Universal Robots URScript: samho_main_Fillet_2024_03_05.script

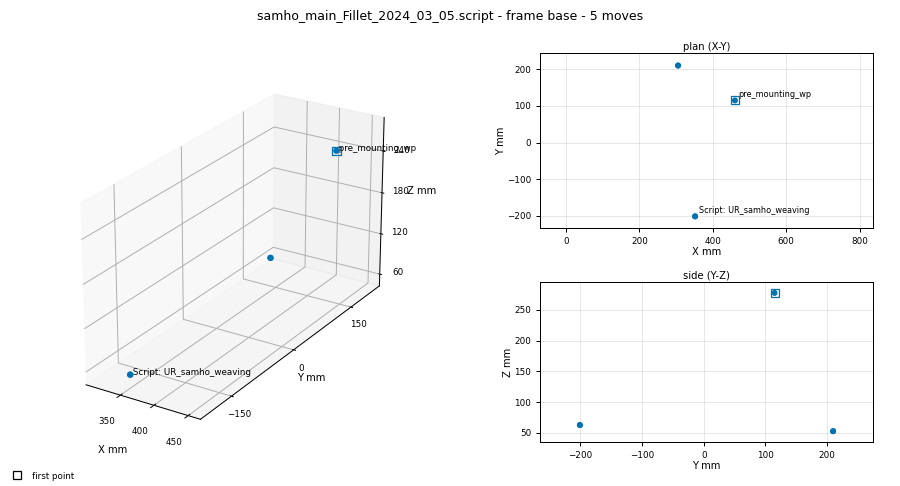
[picture p0: tool path of samho_main_Fillet_2024_03_05.script in frame base, 5 of 126 moves have a stored position in this frame; points joined in program order, loops and branches not executed]
def samho_main_Fillet_2024_03_05():
  modbus_add_signal("127.0.0.1", 255, 239, 2, "MODBUS_1", False)
  modbus_set_signal_update_frequency("MODBUS_1", 1)
  modbus_add_signal("127.0.0.1", 255, 153, 2, "MODBUS_2", False)
  modbus_set_signal_update_frequency("MODBUS_2", 10)
  modbus_add_signal("127.0.0.1", 255, 154, 2, "MODBUS_3", False)
  modbus_set_signal_update_frequency("MODBUS_3", 10)
  modbus_add_signal("127.0.0.1", 255, 204, 2, "MODBUS_4", False)
  modbus_set_signal_update_frequency("MODBUS_4", 10)
  modbus_add_signal("127.0.0.1", 255, 205, 2, "MODBUS_5", False)
  modbus_set_signal_update_frequency("MODBUS_5", 10)
  modbus_add_signal("127.0.0.1", 255, 201, 2, "MODBUS_6", False)
  modbus_set_signal_update_frequency("MODBUS_6", 10)
  modbus_add_signal("127.0.0.1", 255, 202, 2, "MODBUS_7", False)
  modbus_set_signal_update_frequency("MODBUS_7", 10)
  set_tcp(p[-0.20862,-0.00524,0.38449,1.2551,0.019,-2.8747])
  set_payload(2.4, [-0.085, 0.00191, 0.125])
  set_standard_analog_input_domain(0, 1)
  set_standard_analog_input_domain(1, 1)
  set_tool_analog_input_domain(0, 1)
  set_tool_analog_input_domain(1, 1)
  set_analog_outputdomain(0, 1)
  set_analog_outputdomain(1, 1)
  set_input_actions_to_default()
  set_tool_digital_input_action(1, "freedrive")
  set_runstate_standard_digital_outputs([0])
  set_runstate_standard_digital_output_to_value(0, 1)
  set_runstate_standard_digital_output_to_value(7, 3)
  set_gravity([0.0, 0.0, 9.82])
  set_tool_voltage(24)
  set_safety_mode_transition_hardness(1)
  step_count_f2810c44_adc3_46b3_ab5f_e83060e03eab = 0.0
  thread Step_Counter_Thread_7db14191_1226_40d4_95da_5f36167022e0():
    while (True):
      step_count_f2810c44_adc3_46b3_ab5f_e83060e03eab = step_count_f2810c44_adc3_46b3_ab5f_e83060e03eab + 1.0
      sync()
    end
  end
  run Step_Counter_Thread_7db14191_1226_40d4_95da_5f36167022e0()
  global A_Prepos_l=[p[0, 0, 0, 0, 0, 0], p[0, 0, 0, 0, 0, 0], p[0, 0, 0, 0, 0, 0], p[0, 0, 0, 0, 0, 0], p[0, 0, 0, 0, 0, 0], p[0.46809, 0.38153, 0.04984, -2.35756, -1.0346, -1.29868], p[0, 0, 0, 0, 0, 0], p[0.46992, -0.42847, 0.05169, 2.24214, -1.10327, 1.24657], p[0, 0, 0, 0, 0, 0], p[0, 0, 0, 0, 0, 0], p[0, 0, 0, 0, 0, 0], p[0, 0, 0, 0, 0, 0], p[0, 0, 0, 0, 0, 0], p[0, 0, 0, 0, 0, 0], p[0, 0, 0, 0, 0, 0], p[0, 0, 0, 0, 0, 0]]
  global x_offset_3=[0, 0, 0, 0, 0, 0, 0, 0, 0, 0, 0, 0, 0, 0, 0, 0, 0, 0, 0, 0, 0, 0, 0, 0, 0, 0, 0, 0, 0, 0, 0, 0, 0, 0, 0, 0, 0, 0, 0, 0, 0, 0, 0, 0, 0, 0, 0, 0, 0, 0, 0, 0, 0, 0, 0, 0, 0, 0, 0, 0, 0, 0, 0, 0, 0, 0, 0, 0, 0, 0, 0, 0, 0, 0, 0, 0, 0, 0, 0, 0, 0, 0, 0, 0, 0, 0, 0, 0, 0, 0, 0, 0, 0, 0, 0, 0, 0, 0, 0, 0, 0, 0, 0, 0, 0, 0, 0, 0, 0, 0, 0, 0, 0, 0, 0, 0, 0, 0, 0, 0, 0, 0, 0, 0, 0, 0, 0, 0, 0, 0, 0, 0, 0, 0, 0, 0, 0, 0, 0, 0, 0, 0, 0, 0, 0, 0, 0, 0, 0, 0, 0, 0, 0, 0, 0, 0, 0, 0, 0, 0, 0, 0, 0, 0, 0, 0, 0, 0, 0, 0, 0, 0, 0, 0, 0, 0, 0, 0, 0, 0, 0, 0, 0, 0, 0, 0, 0, 0, 0, 0, 0, 0, 0, 0, 0, 0, 0, 0, 0, 0, 0, 0, 0, 0, 0, 0, 0, 0, 0, 0, 0, 0, 0, 0, 0, 0, 0, 0, 0, 0, 0, 0, 0, 0, 0, 0, 0, 0, 0, 0, 0, 0, 0, 0, 0, 0, 0, 0, 0, 0, 0, 0, 0, 0, 0, 0, 0, 0, 0, 0, 0, 0, 0, 0, 0, 0, 0, 0, 0, 0, 0, 0, 0, 0, 0, 0, 0, 0, 0, 0, 0, 0, 0, 0, 0, 0, 0, 0, 0]
  global x_offset_2=[0, 0, 0, 0.0209, 0.0209, 0.0209, 0.0209, 0.02404, 0.02404, 0.02404, 0.67295, 0.67295, 0.67295, 2.17295, 2.17295, 2.17295, 2.71631, 2.71631, 2.71631, 4.21631, 4.21631, 4.70369, 4.70369, 4.70369, 4.88237, 4.88237, 4.88237, 4.71508, 4.71508, 4.71508, 4.94078, 4.94078, 4.79072, 4.79072, 4.79072, 4.75658, 4.75658, 4.75658, 4.91311, 4.91311, 4.91311, 4.93686, 4.93686, 4.93686, 5.14007, 5.14007, 5.1772, 5.1772, 5.1772, 5.18907, 5.18907, 5.18907, 5.23752, 5.23752, 5.23752, 6.44215, 6.44215, 6.47898, 6.47898, 6.47898, 6.4358, 6.4358, 6.4358, 6.27225, 6.27225, 6.27225, 6.28625, 6.28625, 6.28625, 6.32596, 6.32596, 6.09664, 6.09664, 6.09664, 5.90683, 5.90683, 5.90683, 5.8852, 5.8852, 5.8852, 7.21499, 7.21499, 7.23472, 7.23472, 7.23472, 6.60284, 6.60284, 6.60284, 6.76782, 6.76782, 6.76782, 6.77998, 6.77998, 6.77998, 7.28903, 7.28903, 7.28454, 7.28454, 7.28454, 0, 0, 0, 0, 0, 0, 0, 0, 0, 0, 0, 0, 0, 0, 0, 0, 0, 0, 0, 0, 0, 0, 0, 0, 0, 0, 0, 0, 0, 0, 0, 0, 0, 0, 0, 0, 0, 0, 0, 0, 0, 0, 0, 0, 0, 0, 0, 0, 0, 0, 0, 0, 0, 0, 0, 0, 0, 0, 0, 0, 0, 0, 0, 0, 0, 0, 0, 0, 0, 0, 0, 0, 0, 0, 0, 0, 0, 0, 0, 0, 0, 0, 0, 0, 0, 0, 0, 0, 0, 0, 0, 0, 0, 0, 0, 0, 0, 0, 0, 0, 0, 0, 0, 0, 0, 0, 0, 0, 0, 0, 0, 0, 0, 0, 0, 0, 0, 0, 0, 0, 0, 0, 0, 0, 0, 0, 0, 0, 0, 0, 0, 0, 0, 0, 0, 0, 0, 0, 0, 0, 0, 0, 0, 0, 0, 0, 0, 0, 0, 0, 0, 0, 0, 0, 0, 0, 0, 0, 0, 0, 0, 0, 0, 0, 0, 0, 0, 0, 0, 0, 0, 0, 0, 0, 0, 0, 0, 0, 0, 0]
  global A_Distance_list=[0, 0, 0, 0, 0, 0, 0, 0, 0, 0, 0, 0, 0, 0, 0, 0]
  global x_offset_1=[0, 0, 0, -0.02252, -0.02252, -0.02252, -0.02252, 0.13096, 0.13096, 0.13096, 2.13096, 2.13096, 2.13096, 2.79881, 2.79881, 2.79881, 2.79282, 2.79282, 2.79282, 2.61839, 2.61839, 2.63263, 2.63263, 2.63263, 2.62365, 2.62365, 2.62365, 3.30637, 3.30637, 3.30637, 4.74748, 4.74748, 4.71042, 4.71042, 4.71042, 4.68978, 4.68978, 4.68978, 4.48892, 4.48892, 4.48892, 3.24306, 3.24306, 3.24306, 3.21841, 3.21841, 3.25956, 3.25956, 3.25956, 5.25956, 5.25956, 5.25956, 5.09671, 5.09671, 5.09671, 5.11266, 5.11266, 4.90289, 4.90289, 4.90289, 4.02534, 4.02534, 4.02534, 4.19985, 4.19985, 4.19985, 4.03315, 4.03315, 4.03315, 4.03825, 4.03825, 4.0859, 4.0859, 4.0859, 4.12182, 4.12182, 4.12182, 5.56392, 5.56392, 5.56392, 5.61278, 5.61278, 5.56799, 5.56799, 5.56799, 6.3781, 6.3781, 6.3781, 5.52948, 5.52948, 5.52948, 5.5349, 5.5349, 5.5349, 5.52338, 5.52338, 6.3895, 6.3895, 6.3895, 0, 0, 0, 0, 0, 0, 0, 0, 0, 0, 0, 0, 0, 0, 0, 0, 0, 0, 0, 0, 0, 0, 0, 0, 0, 0, 0, 0, 0, 0, 0, 0, 0, 0, 0, 0, 0, 0, 0, 0, 0, 0, 0, 0, 0, 0, 0, 0, 0, 0, 0, 0, 0, 0, 0, 0, 0, 0, 0, 0, 0, 0, 0, 0, 0, 0, 0, 0, 0, 0, 0, 0, 0, 0, 0, 0, 0, 0, 0, 0, 0, 0, 0, 0, 0, 0, 0, 0, 0, 0, 0, 0, 0, 0, 0, 0, 0, 0, 0, 0, 0, 0, 0, 0, 0, 0, 0, 0, 0, 0, 0, 0, 0, 0, 0, 0, 0, 0, 0, 0, 0, 0, 0, 0, 0, 0, 0, 0, 0, 0, 0, 0, 0, 0, 0, 0, 0, 0, 0, 0, 0, 0, 0, 0, 0, 0, 0, 0, 0, 0, 0, 0, 0, 0, 0, 0, 0, 0, 0, 0, 0, 0, 0, 0, 0, 0, 0, 0, 0, 0, 0, 0, 0, 0, 0, 0, 0, 0, 0, 0]
  global last_tilt_deg=[30, -0, 0]
  global step_2f=2
  global A_touch_bottom=p[0.4884, 0.0279, -0.05448, 2.85052, -0.02454, 1.30656]
  global A_Touch_trig_l=[False, False, False, False, False, True, False, True, False, False, False]
  global Auto_trig=True
  global Auto_W_num=[31, 32, 41, 42, 51, 52, 0, 0, 0, 0, 0, 0, 0, 0, 0]
  global Reset_Trig=False
  global last_wv_wp1=p[0.48809, -0.02364, -0.05448, 2.88623, -0.01704, 1.22388]
  global A_Speed_list=[0, 0, 0, 0, 0, 0, 0, 0, 0, 0, 0, 0, 0, 0, 0, 0]
  global last_z_bottom=-0.0502
  global A_Touch_p=[p[0, 0, 0, 0, 0, 0], p[0, 0, 0, 0, 0, 0], p[0, 0, 0, 0, 0, 0], p[0, 0, 0, 0, 0, 0], p[0, 0, 0, 0, 0, 0], p[0.49492, 0.37647, -0.00373, -1.74067, 1.76135, -0.74873], p[0, 0, 0, 0, 0, 0], p[0.49325, -0.42377, 0.00921, -1.77678, 1.78638, -0.71819], p[0, 0, 0, 0, 0, 0], p[0, 0, 0, 0, 0, 0], p[0, 0, 0, 0, 0, 0], p[0, 0, 0, 0, 0, 0], p[0, 0, 0, 0, 0, 0], p[0, 0, 0, 0, 0, 0], p[0, 0, 0, 0, 0, 0], p[0, 0, 0, 0, 0, 0]]
  global z_offset_3=[0, 0, 0, 0, 0, 0, 0, 0, 0, 0, 0, 0, 0, 0, 0, 0, 0, 0, 0, 0, 0, 0, 0, 0, 0, 0, 0, 0, 0, 0, 0, 0, 0, 0, 0, 0, 0, 0, 0, 0, 0, 0, 0, 0, 0, 0, 0, 0, 0, 0, 0, 0, 0, 0, 0, 0, 0, 0, 0, 0, 0, 0, 0, 0, 0, 0, 0, 0, 0, 0, 0, 0, 0, 0, 0, 0, 0, 0, 0, 0, 0, 0, 0, 0, 0, 0, 0, 0, 0, 0, 0, 0, 0, 0, 0, 0, 0, 0, 0, 0, 0, 0, 0, 0, 0, 0, 0, 0, 0, 0, 0, 0, 0, 0, 0, 0, 0, 0, 0, 0, 0, 0, 0, 0, 0, 0, 0, 0, 0, 0, 0, 0, 0, 0, 0, 0, 0, 0, 0, 0, 0, 0, 0, 0, 0, 0, 0, 0, 0, 0, 0, 0, 0, 0, 0, 0, 0, 0, 0, 0, 0, 0, 0, 0, 0, 0, 0, 0, 0, 0, 0, 0, 0, 0, 0, 0, 0, 0, 0, 0, 0, 0, 0, 0, 0, 0, 0, 0, 0, 0, 0, 0, 0, 0, 0, 0, 0, 0, 0, 0, 0, 0, 0, 0, 0, 0, 0, 0, 0, 0, 0, 0, 0, 0, 0, 0, 0, 0, 0, 0, 0, 0, 0, 0, 0, 0, 0, 0, 0, 0, 0, 0, 0, 0, 0, 0, 0, 0, 0, 0, 0, 0, 0, 0, 0, 0, 0, 0, 0, 0, 0, 0, 0, 0, 0, 0, 0, 0, 0, 0, 0, 0, 0, 0, 0, 0, 0, 0, 0, 0, 0, 0, 0, 0, 0, 0, 0, 0, 0]
  global z_offset_2=[0, 0, 0, 0.77652, 0.77652, 0.77652, 0.77652, 4.77652, 4.77652, 4.77652, 8.77652, 8.77652, 8.77652, 9.70696, 9.70696, 9.70696, 9.70696, 9.70696, 9.70696, 9.86322, 9.86322, 11.04005, 11.04005, 11.04005, 11.70378, 11.70378, 11.70378, 12.6435, 12.6435, 12.6435, 12.8145, 12.8145, 13.44251, 13.44251, 13.44251, 14.37812, 14.37812, 14.37812, 14.43959, 14.43959, 14.43959, 14.63644, 14.63644, 14.63644, 14.76133, 14.76133, 16.3973, 16.3973, 16.3973, 17.51846, 17.51846, 17.51846, 17.46024, 17.46024, 17.46024, 16.57938, 16.57938, 15.57852, 15.57852, 15.57852, 14.06174, 14.06174, 14.06174, 13.91328, 13.91328, 13.91328, 14.75741, 14.75741, 14.75741, 14.95018, 14.95018, 14.9305, 14.9305, 14.9305, 14.91085, 14.91085, 14.91085, 13.42972, 13.42972, 13.42972, 12.56827, 12.56827, 11.94768, 11.94768, 11.94768, 11.06049, 11.06049, 11.06049, 10.36556, 10.36556, 10.36556, 9.66223, 9.66223, 9.66223, 8.10136, 8.10136, 4.45952, 4.45952, 4.45952, 0, 0, 0, 0, 0, 0, 0, 0, 0, 0, 0, 0, 0, 0, 0, 0, 0, 0, 0, 0, 0, 0, 0, 0, 0, 0, 0, 0, 0, 0, 0, 0, 0, 0, 0, 0, 0, 0, 0, 0, 0, 0, 0, 0, 0, 0, 0, 0, 0, 0, 0, 0, 0, 0, 0, 0, 0, 0, 0, 0, 0, 0, 0, 0, 0, 0, 0, 0, 0, 0, 0, 0, 0, 0, 0, 0, 0, 0, 0, 0, 0, 0, 0, 0, 0, 0, 0, 0, 0, 0, 0, 0, 0, 0, 0, 0, 0, 0, 0, 0, 0, 0, 0, 0, 0, 0, 0, 0, 0, 0, 0, 0, 0, 0, 0, 0, 0, 0, 0, 0, 0, 0, 0, 0, 0, 0, 0, 0, 0, 0, 0, 0, 0, 0, 0, 0, 0, 0, 0, 0, 0, 0, 0, 0, 0, 0, 0, 0, 0, 0, 0, 0, 0, 0, 0, 0, 0, 0, 0, 0, 0, 0, 0, 0, 0, 0, 0, 0, 0, 0, 0, 0, 0, 0, 0, 0, 0, 0, 0, 0]
  global z_offset_1=[0, 0, 0, 3.84239, 3.84239, 3.84239, 3.84239, 7.76295, 7.76295, 7.76295, 7.92335, 7.92335, 7.92335, 8.7083, 8.7083, 8.7083, 9.56251, 9.56251, 9.56251, 11.37986, 11.37986, 13.17871, 13.17871, 13.17871, 14.66928, 14.66928, 14.66928, 14.80578, 14.80578, 14.80578, 14.83719, 14.83719, 15.63828, 15.63828, 15.63828, 15.72912, 15.72912, 15.72912, 15.59233, 15.59233, 15.59233, 15.55065, 15.55065, 15.55065, 17.0551, 17.0551, 20.57114, 20.57114, 20.57114, 20.52132, 20.52132, 20.52132, 19.36419, 19.36419, 19.36419, 19.2215, 19.2215, 19.17005, 19.17005, 19.17005, 18.97372, 18.97372, 18.97372, 18.80152, 18.80152, 18.80152, 19.52527, 19.52527, 19.52527, 19.70213, 19.70213, 19.80342, 19.80342, 19.80342, 18.96513, 18.96513, 18.96513, 17.54204, 17.54204, 17.54204, 16.80619, 16.80619, 13.73593, 13.73593, 13.73593, 13.62525, 13.62525, 13.62525, 12.71187, 12.71187, 12.71187, 11.52228, 11.52228, 11.52228, 9.66149, 9.66149, 9.49537, 9.49537, 9.49537, 0, 0, 0, 0, 0, 0, 0, 0, 0, 0, 0, 0, 0, 0, 0, 0, 0, 0, 0, 0, 0, 0, 0, 0, 0, 0, 0, 0, 0, 0, 0, 0, 0, 0, 0, 0, 0, 0, 0, 0, 0, 0, 0, 0, 0, 0, 0, 0, 0, 0, 0, 0, 0, 0, 0, 0, 0, 0, 0, 0, 0, 0, 0, 0, 0, 0, 0, 0, 0, 0, 0, 0, 0, 0, 0, 0, 0, 0, 0, 0, 0, 0, 0, 0, 0, 0, 0, 0, 0, 0, 0, 0, 0, 0, 0, 0, 0, 0, 0, 0, 0, 0, 0, 0, 0, 0, 0, 0, 0, 0, 0, 0, 0, 0, 0, 0, 0, 0, 0, 0, 0, 0, 0, 0, 0, 0, 0, 0, 0, 0, 0, 0, 0, 0, 0, 0, 0, 0, 0, 0, 0, 0, 0, 0, 0, 0, 0, 0, 0, 0, 0, 0, 0, 0, 0, 0, 0, 0, 0, 0, 0, 0, 0, 0, 0, 0, 0, 0, 0, 0, 0, 0, 0, 0, 0, 0, 0, 0, 0, 0]
  global last_wv_line=p[0.49409, -0.02365, -0.05448, -1.74067, 1.76135, -0.74873]
  global last_pose=p[0.50354, -0.16852, -0.0383, 2.73154, -0.12092, 1.1572]
  global Auto_total_cell=6
  global Auto_cur_cell=3
  global Base=p[0.0,0.0,0.0,0.0,0.0,0.0]
  global save_timer=0
  global timer_1=0
  def calculate_point_to_move_towards(feature, direction, position_distance):
    local posDir=[direction[0], direction[1], direction[2]]
    if (norm(posDir) < 1e-6):
      return get_target_waypoint()
    end
    local direction_vector_normalized=normalize(posDir)
    local displacement_pose=p[direction_vector_normalized[0] * position_distance,direction_vector_normalized[1] * position_distance,direction_vector_normalized[2] * position_distance,0,0,0]
    local wanted_displacement_in_base_frame=pose_sub(pose_trans(feature, displacement_pose), feature)
    return pose_add(get_target_waypoint(), wanted_displacement_in_base_frame)
  end
  global save_timer_is_counting=False
  global timer_1_is_counting=False
  thread Timer_Thread():
    while (True):
      if (save_timer_is_counting):
        save_timer = save_timer + get_steptime()
      end
      if (timer_1_is_counting):
        timer_1 = timer_1 + get_steptime()
      end
      sync()
    end
  end
  run Timer_Thread()
  def cell_info():
    $ 1549 "cell_info" "noBreak"
    $ 1550 "'cell_setting'"
    # 'cell_setting'
    $ 1551 "a7_f_distance≔get_center"
    global a7_f_distance=get_center
    $ 1552 "'dis + 125'"
    # 'dis + 125'
    $ 1553 "If simulation_mode"
    if (simulation_mode):
      $ 1554 "a6_f_height_l≔190"
      global a6_f_height_l=190
      $ 1555 "a6_f_height_r≔190"
      global a6_f_height_r=190
      $ 1556 "a6_f_width≔690"
      global a6_f_width=690
      $ 1557 "a6_callar_hor≔100"
      global a6_callar_hor=100
      $ 1558 "a6_callar_vert≔100"
      global a6_callar_vert=100
      $ 1559 "center_height≔50"
      global center_height=50
      $ 1560 "EXT_flag1≔integer_to_binary_list(2048)"
      global EXT_flag1= integer_to_binary_list (2048)
      $ 1561 "get_margin_z≔50"
      global get_margin_z=50
    else:
      $ 1562 "Else" "noBreak"
      $ 1563 "a6_f_height_l≔read_port_register(173)"
      global a6_f_height_l= read_port_register (173)
      $ 1564 "a6_f_height_r≔read_port_register(174)"
      global a6_f_height_r= read_port_register (174)
      $ 1565 "a6_f_width≔read_port_register(175)"
      global a6_f_width= read_port_register (175)
      $ 1566 "a6_callar_hor≔read_port_register(181)"
      global a6_callar_hor= read_port_register (181)
      $ 1567 "a6_callar_vert≔read_port_register(182)"
      global a6_callar_vert= read_port_register (182)
      $ 1568 "center_height≔read_port_register(237)"
      global center_height=read_port_register(237)
      $ 1569 "EXT_flag1≔integer_to_binary_list(read_port_register(179))"
      global EXT_flag1= integer_to_binary_list ( read_port_register (179))
      $ 1571 "get_margin_z≔read_port_register(238)"
      global get_margin_z=read_port_register(238)
      $ 1573 "If center_height>32765"
      if (center_height>32765):
        $ 1574 "center_height≔center_height-65535"
        global center_height=center_height-65535
      end
      $ 1575 "If get_margin_z>32765"
      if (get_margin_z>32765):
        $ 1576 "get_margin_z≔get_margin_z-65535"
        global get_margin_z=get_margin_z-65535
      end
    end
    $ 1577 "Initialization"
    $ 1578 "CELL_ROBOT_DIST≔a7_f_distance"
    global CELL_ROBOT_DIST=a7_f_distance
    $ 1579 "CELL_WIDTH≔a6_f_width"
    global CELL_WIDTH=a6_f_width
  end
  def robotand_cell_initalizat():
    $ 1580 "robotand_cell_initalizat" "noBreak"
    $ 1581 "If Auto_trig≟ True "
    if (Auto_trig ==   True  ):
      $ 1582 "Auto_trig≔ False "
      global Auto_trig=  False
      $ 1583 "init"
      $ 1584 "write_port_register(cell_3f_2f_151,0)"
      write_port_register(cell_3f_2f_151,0)
      $ 1585 "write_port_register(cell_info_152,0)"
      write_port_register(cell_info_152,0)
      $ 1586 "write_port_register(weld_req_153,0)"
      write_port_register(weld_req_153,0)
      $ 1587 "write_port_register(touch_cell_155,0)"
      write_port_register(touch_cell_155,0)
      $ 1588 "write_port_register(touch_num_156,0)"
      write_port_register(touch_num_156,0)
      $ 1589 "write_port_register(touch_done_157,0)"
      write_port_register(touch_done_157,0)
      $ 1590 "write_port_register(weld_done_137,0)"
      write_port_register(weld_done_137,0)
      $ 1591 "write_port_register(135,0)"
      write_port_register(135,0)
      $ 1592 "write_port_register(136,0)"
      write_port_register(136,0)
      $ 1593 "write_port_register(165,0)"
      write_port_register(165,0)
      $ 1594 "write_port_register(166,0)"
      write_port_register(166,0)
      $ 1595 "write_port_register(167,0)"
      write_port_register(167,0)
      $ 1596 "write_port_register(169,0)"
      write_port_register(169,0)
      $ 1597 "write_port_register(170,0)"
      write_port_register(170,0)
      $ 1598 "write_port_register(221,0)"
      write_port_register(221,0)
      $ 1599 "write_port_register(222,0)"
      write_port_register(222,0)
      $ 1600 "write_port_register(223,0)"
      write_port_register(223,0)
      $ 1601 "write_port_register(224,0)"
      write_port_register(224,0)
      $ 1602 "write_port_register(225,0)"
      write_port_register(225,0)
      $ 1603 "write_port_register(226,0)"
      write_port_register(226,0)
      $ 1604 "write_port_register(227,0)"
      write_port_register(227,0)
      $ 1605 "write_port_register(228,0)"
      write_port_register(228,0)
      $ 1606 "write_port_register(240,0)"
      write_port_register(240,0)
      $ 1607 "write_port_register(176,0)"
      write_port_register(176,0)
      $ 1608 "write_port_register(177,0)"
      write_port_register(177,0)
      $ 1609 "write_port_register(154,0)"
      write_port_register(154,0)
    end
    $ 1610 "sync()"
    sync()
  end
  def reset_multi_record():
    $ 1611 "reset_multi_record" "noBreak"
    $ 1612 "step_2f≔0"
    global step_2f=0
    $ 1613 "x_offset_1≔[0, 0, 0, 0, 0, 0, 0, 0, 0, 0, 0, 0, 0, 0, 0, 0, 0, 0, 0, 0, 0, 0, 0, 0, 0, 0, 0, 0, 0, 0, 0, 0, 0, 0, 0, 0, 0, 0, 0, 0, 0, 0, 0, 0, 0, 0, 0, 0, 0, 0, 0, 0, 0, 0, 0, 0, 0, 0, 0, 0, 0, 0, 0, 0, 0, 0, 0, 0, 0, 0, 0, 0, 0, 0, 0, 0, 0, 0, 0, 0, 0, 0, 0, 0, 0, 0, 0, 0, 0, 0, 0, 0, 0, 0, 0, 0, 0, 0, 0, 0, 0, 0, 0, 0, 0, 0, 0, 0, 0, 0, 0, 0, 0, 0, 0, 0, 0, 0, 0, 0, 0, 0, 0, 0, 0, 0, 0, 0, 0, 0, 0, 0, 0, 0, 0, 0, 0, 0, 0, 0, 0, 0, 0, 0, 0, 0, 0, 0, 0, 0, 0, 0, 0, 0, 0, 0, 0, 0, 0, 0, 0, 0, 0, 0, 0, 0, 0, 0, 0, 0, 0, 0, 0, 0, 0, 0, 0, 0, 0, 0, 0, 0, 0, 0, 0, 0, 0, 0, 0, 0, 0, 0, 0, 0, 0, 0, 0, 0, 0, 0, 0, 0, 0, 0, 0, 0, 0, 0, 0, 0, 0, 0, 0, 0, 0, 0, 0, 0, 0, 0, 0, 0, 0, 0, 0, 0, 0, 0, 0, 0, 0, 0, 0, 0, 0, 0, 0, 0, 0, 0, 0, 0, 0, 0, 0, 0, 0, 0, 0, 0, 0, 0, 0, 0, 0, 0, 0, 0, 0, 0, 0, 0, 0, 0, 0, 0, 0, 0, 0, 0, 0, 0, 0, 0, 0, 0, 0, 0, 0]"
    global x_offset_1=[0, 0, 0, 0, 0, 0, 0, 0, 0, 0, 0, 0, 0, 0, 0, 0, 0, 0, 0, 0, 0, 0, 0, 0, 0, 0, 0, 0, 0, 0, 0, 0, 0, 0, 0, 0, 0, 0, 0, 0, 0, 0, 0, 0, 0, 0, 0, 0, 0, 0, 0, 0, 0, 0, 0, 0, 0, 0, 0, 0, 0, 0, 0, 0, 0, 0, 0, 0, 0, 0, 0, 0, 0, 0, 0, 0, 0, 0, 0, 0, 0, 0, 0, 0, 0, 0, 0, 0, 0, 0, 0, 0, 0, 0, 0, 0, 0, 0, 0, 0, 0, 0, 0, 0, 0, 0, 0, 0, 0, 0, 0, 0, 0, 0, 0, 0, 0, 0, 0, 0, 0, 0, 0, 0, 0, 0, 0, 0, 0, 0, 0, 0, 0, 0, 0, 0, 0, 0, 0, 0, 0, 0, 0, 0, 0, 0, 0, 0, 0, 0, 0, 0, 0, 0, 0, 0, 0, 0, 0, 0, 0, 0, 0, 0, 0, 0, 0, 0, 0, 0, 0, 0, 0, 0, 0, 0, 0, 0, 0, 0, 0, 0, 0, 0, 0, 0, 0, 0, 0, 0, 0, 0, 0, 0, 0, 0, 0, 0, 0, 0, 0, 0, 0, 0, 0, 0, 0, 0, 0, 0, 0, 0, 0, 0, 0, 0, 0, 0, 0, 0, 0, 0, 0, 0, 0, 0, 0, 0, 0, 0, 0, 0, 0, 0, 0, 0, 0, 0, 0, 0, 0, 0, 0, 0, 0, 0, 0, 0, 0, 0, 0, 0, 0, 0, 0, 0, 0, 0, 0, 0, 0, 0, 0, 0, 0, 0, 0, 0, 0, 0, 0, 0, 0, 0, 0, 0, 0, 0, 0]
    $ 1614 "x_offset_2≔[0, 0, 0, 0, 0, 0, 0, 0, 0, 0, 0, 0, 0, 0, 0, 0, 0, 0, 0, 0, 0, 0, 0, 0, 0, 0, 0, 0, 0, 0, 0, 0, 0, 0, 0, 0, 0, 0, 0, 0, 0, 0, 0, 0, 0, 0, 0, 0, 0, 0, 0, 0, 0, 0, 0, 0, 0, 0, 0, 0, 0, 0, 0, 0, 0, 0, 0, 0, 0, 0, 0, 0, 0, 0, 0, 0, 0, 0, 0, 0, 0, 0, 0, 0, 0, 0, 0, 0, 0, 0, 0, 0, 0, 0, 0, 0, 0, 0, 0, 0, 0, 0, 0, 0, 0, 0, 0, 0, 0, 0, 0, 0, 0, 0, 0, 0, 0, 0, 0, 0, 0, 0, 0, 0, 0, 0, 0, 0, 0, 0, 0, 0, 0, 0, 0, 0, 0, 0, 0, 0, 0, 0, 0, 0, 0, 0, 0, 0, 0, 0, 0, 0, 0, 0, 0, 0, 0, 0, 0, 0, 0, 0, 0, 0, 0, 0, 0, 0, 0, 0, 0, 0, 0, 0, 0, 0, 0, 0, 0, 0, 0, 0, 0, 0, 0, 0, 0, 0, 0, 0, 0, 0, 0, 0, 0, 0, 0, 0, 0, 0, 0, 0, 0, 0, 0, 0, 0, 0, 0, 0, 0, 0, 0, 0, 0, 0, 0, 0, 0, 0, 0, 0, 0, 0, 0, 0, 0, 0, 0, 0, 0, 0, 0, 0, 0, 0, 0, 0, 0, 0, 0, 0, 0, 0, 0, 0, 0, 0, 0, 0, 0, 0, 0, 0, 0, 0, 0, 0, 0, 0, 0, 0, 0, 0, 0, 0, 0, 0, 0, 0, 0, 0, 0, 0, 0, 0, 0, 0, 0]"
    global x_offset_2=[0, 0, 0, 0, 0, 0, 0, 0, 0, 0, 0, 0, 0, 0, 0, 0, 0, 0, 0, 0, 0, 0, 0, 0, 0, 0, 0, 0, 0, 0, 0, 0, 0, 0, 0, 0, 0, 0, 0, 0, 0, 0, 0, 0, 0, 0, 0, 0, 0, 0, 0, 0, 0, 0, 0, 0, 0, 0, 0, 0, 0, 0, 0, 0, 0, 0, 0, 0, 0, 0, 0, 0, 0, 0, 0, 0, 0, 0, 0, 0, 0, 0, 0, 0, 0, 0, 0, 0, 0, 0, 0, 0, 0, 0, 0, 0, 0, 0, 0, 0, 0, 0, 0, 0, 0, 0, 0, 0, 0, 0, 0, 0, 0, 0, 0, 0, 0, 0, 0, 0, 0, 0, 0, 0, 0, 0, 0, 0, 0, 0, 0, 0, 0, 0, 0, 0, 0, 0, 0, 0, 0, 0, 0, 0, 0, 0, 0, 0, 0, 0, 0, 0, 0, 0, 0, 0, 0, 0, 0, 0, 0, 0, 0, 0, 0, 0, 0, 0, 0, 0, 0, 0, 0, 0, 0, 0, 0, 0, 0, 0, 0, 0, 0, 0, 0, 0, 0, 0, 0, 0, 0, 0, 0, 0, 0, 0, 0, 0, 0, 0, 0, 0, 0, 0, 0, 0, 0, 0, 0, 0, 0, 0, 0, 0, 0, 0, 0, 0, 0, 0, 0, 0, 0, 0, 0, 0, 0, 0, 0, 0, 0, 0, 0, 0, 0, 0, 0, 0, 0, 0, 0, 0, 0, 0, 0, 0, 0, 0, 0, 0, 0, 0, 0, 0, 0, 0, 0, 0, 0, 0, 0, 0, 0, 0, 0, 0, 0, 0, 0, 0, 0, 0, 0, 0, 0, 0, 0, 0, 0]
    $ 1615 "x_offset_3≔[0, 0, 0, 0, 0, 0, 0, 0, 0, 0, 0, 0, 0, 0, 0, 0, 0, 0, 0, 0, 0, 0, 0, 0, 0, 0, 0, 0, 0, 0, 0, 0, 0, 0, 0, 0, 0, 0, 0, 0, 0, 0, 0, 0, 0, 0, 0, 0, 0, 0, 0, 0, 0, 0, 0, 0, 0, 0, 0, 0, 0, 0, 0, 0, 0, 0, 0, 0, 0, 0, 0, 0, 0, 0, 0, 0, 0, 0, 0, 0, 0, 0, 0, 0, 0, 0, 0, 0, 0, 0, 0, 0, 0, 0, 0, 0, 0, 0, 0, 0, 0, 0, 0, 0, 0, 0, 0, 0, 0, 0, 0, 0, 0, 0, 0, 0, 0, 0, 0, 0, 0, 0, 0, 0, 0, 0, 0, 0, 0, 0, 0, 0, 0, 0, 0, 0, 0, 0, 0, 0, 0, 0, 0, 0, 0, 0, 0, 0, 0, 0, 0, 0, 0, 0, 0, 0, 0, 0, 0, 0, 0, 0, 0, 0, 0, 0, 0, 0, 0, 0, 0, 0, 0, 0, 0, 0, 0, 0, 0, 0, 0, 0, 0, 0, 0, 0, 0, 0, 0, 0, 0, 0, 0, 0, 0, 0, 0, 0, 0, 0, 0, 0, 0, 0, 0, 0, 0, 0, 0, 0, 0, 0, 0, 0, 0, 0, 0, 0, 0, 0, 0, 0, 0, 0, 0, 0, 0, 0, 0, 0, 0, 0, 0, 0, 0, 0, 0, 0, 0, 0, 0, 0, 0, 0, 0, 0, 0, 0, 0, 0, 0, 0, 0, 0, 0, 0, 0, 0, 0, 0, 0, 0, 0, 0, 0, 0, 0, 0, 0, 0, 0, 0, 0, 0, 0, 0, 0, 0, 0]"
    global x_offset_3=[0, 0, 0, 0, 0, 0, 0, 0, 0, 0, 0, 0, 0, 0, 0, 0, 0, 0, 0, 0, 0, 0, 0, 0, 0, 0, 0, 0, 0, 0, 0, 0, 0, 0, 0, 0, 0, 0, 0, 0, 0, 0, 0, 0, 0, 0, 0, 0, 0, 0, 0, 0, 0, 0, 0, 0, 0, 0, 0, 0, 0, 0, 0, 0, 0, 0, 0, 0, 0, 0, 0, 0, 0, 0, 0, 0, 0, 0, 0, 0, 0, 0, 0, 0, 0, 0, 0, 0, 0, 0, 0, 0, 0, 0, 0, 0, 0, 0, 0, 0, 0, 0, 0, 0, 0, 0, 0, 0, 0, 0, 0, 0, 0, 0, 0, 0, 0, 0, 0, 0, 0, 0, 0, 0, 0, 0, 0, 0, 0, 0, 0, 0, 0, 0, 0, 0, 0, 0, 0, 0, 0, 0, 0, 0, 0, 0, 0, 0, 0, 0, 0, 0, 0, 0, 0, 0, 0, 0, 0, 0, 0, 0, 0, 0, 0, 0, 0, 0, 0, 0, 0, 0, 0, 0, 0, 0, 0, 0, 0, 0, 0, 0, 0, 0, 0, 0, 0, 0, 0, 0, 0, 0, 0, 0, 0, 0, 0, 0, 0, 0, 0, 0, 0, 0, 0, 0, 0, 0, 0, 0, 0, 0, 0, 0, 0, 0, 0, 0, 0, 0, 0, 0, 0, 0, 0, 0, 0, 0, 0, 0, 0, 0, 0, 0, 0, 0, 0, 0, 0, 0, 0, 0, 0, 0, 0, 0, 0, 0, 0, 0, 0, 0, 0, 0, 0, 0, 0, 0, 0, 0, 0, 0, 0, 0, 0, 0, 0, 0, 0, 0, 0, 0, 0, 0, 0, 0, 0, 0, 0]
    $ 1616 "z_offset_1≔[0, 0, 0, 0, 0, 0, 0, 0, 0, 0, 0, 0, 0, 0, 0, 0, 0, 0, 0, 0, 0, 0, 0, 0, 0, 0, 0, 0, 0, 0, 0, 0, 0, 0, 0, 0, 0, 0, 0, 0, 0, 0, 0, 0, 0, 0, 0, 0, 0, 0, 0, 0, 0, 0, 0, 0, 0, 0, 0, 0, 0, 0, 0, 0, 0, 0, 0, 0, 0, 0, 0, 0, 0, 0, 0, 0, 0, 0, 0, 0, 0, 0, 0, 0, 0, 0, 0, 0, 0, 0, 0, 0, 0, 0, 0, 0, 0, 0, 0, 0, 0, 0, 0, 0, 0, 0, 0, 0, 0, 0, 0, 0, 0, 0, 0, 0, 0, 0, 0, 0, 0, 0, 0, 0, 0, 0, 0, 0, 0, 0, 0, 0, 0, 0, 0, 0, 0, 0, 0, 0, 0, 0, 0, 0, 0, 0, 0, 0, 0, 0, 0, 0, 0, 0, 0, 0, 0, 0, 0, 0, 0, 0, 0, 0, 0, 0, 0, 0, 0, 0, 0, 0, 0, 0, 0, 0, 0, 0, 0, 0, 0, 0, 0, 0, 0, 0, 0, 0, 0, 0, 0, 0, 0, 0, 0, 0, 0, 0, 0, 0, 0, 0, 0, 0, 0, 0, 0, 0, 0, 0, 0, 0, 0, 0, 0, 0, 0, 0, 0, 0, 0, 0, 0, 0, 0, 0, 0, 0, 0, 0, 0, 0, 0, 0, 0, 0, 0, 0, 0, 0, 0, 0, 0, 0, 0, 0, 0, 0, 0, 0, 0, 0, 0, 0, 0, 0, 0, 0, 0, 0, 0, 0, 0, 0, 0, 0, 0, 0, 0, 0, 0, 0, 0, 0, 0, 0, 0, 0, 0]"
    global z_offset_1=[0, 0, 0, 0, 0, 0, 0, 0, 0, 0, 0, 0, 0, 0, 0, 0, 0, 0, 0, 0, 0, 0, 0, 0, 0, 0, 0, 0, 0, 0, 0, 0, 0, 0, 0, 0, 0, 0, 0, 0, 0, 0, 0, 0, 0, 0, 0, 0, 0, 0, 0, 0, 0, 0, 0, 0, 0, 0, 0, 0, 0, 0, 0, 0, 0, 0, 0, 0, 0, 0, 0, 0, 0, 0, 0, 0, 0, 0, 0, 0, 0, 0, 0, 0, 0, 0, 0, 0, 0, 0, 0, 0, 0, 0, 0, 0, 0, 0, 0, 0, 0, 0, 0, 0, 0, 0, 0, 0, 0, 0, 0, 0, 0, 0, 0, 0, 0, 0, 0, 0, 0, 0, 0, 0, 0, 0, 0, 0, 0, 0, 0, 0, 0, 0, 0, 0, 0, 0, 0, 0, 0, 0, 0, 0, 0, 0, 0, 0, 0, 0, 0, 0, 0, 0, 0, 0, 0, 0, 0, 0, 0, 0, 0, 0, 0, 0, 0, 0, 0, 0, 0, 0, 0, 0, 0, 0, 0, 0, 0, 0, 0, 0, 0, 0, 0, 0, 0, 0, 0, 0, 0, 0, 0, 0, 0, 0, 0, 0, 0, 0, 0, 0, 0, 0, 0, 0, 0, 0, 0, 0, 0, 0, 0, 0, 0, 0, 0, 0, 0, 0, 0, 0, 0, 0, 0, 0, 0, 0, 0, 0, 0, 0, 0, 0, 0, 0, 0, 0, 0, 0, 0, 0, 0, 0, 0, 0, 0, 0, 0, 0, 0, 0, 0, 0, 0, 0, 0, 0, 0, 0, 0, 0, 0, 0, 0, 0, 0, 0, 0, 0, 0, 0, 0, 0, 0, 0, 0, 0, 0]
    $ 1617 "z_offset_2≔[0, 0, 0, 0, 0, 0, 0, 0, 0, 0, 0, 0, 0, 0, 0, 0, 0, 0, 0, 0, 0, 0, 0, 0, 0, 0, 0, 0, 0, 0, 0, 0, 0, 0, 0, 0, 0, 0, 0, 0, 0, 0, 0, 0, 0, 0, 0, 0, 0, 0, 0, 0, 0, 0, 0, 0, 0, 0, 0, 0, 0, 0, 0, 0, 0, 0, 0, 0, 0, 0, 0, 0, 0, 0, 0, 0, 0, 0, 0, 0, 0, 0, 0, 0, 0, 0, 0, 0, 0, 0, 0, 0, 0, 0, 0, 0, 0, 0, 0, 0, 0, 0, 0, 0, 0, 0, 0, 0, 0, 0, 0, 0, 0, 0, 0, 0, 0, 0, 0, 0, 0, 0, 0, 0, 0, 0, 0, 0, 0, 0, 0, 0, 0, 0, 0, 0, 0, 0, 0, 0, 0, 0, 0, 0, 0, 0, 0, 0, 0, 0, 0, 0, 0, 0, 0, 0, 0, 0, 0, 0, 0, 0, 0, 0, 0, 0, 0, 0, 0, 0, 0, 0, 0, 0, 0, 0, 0, 0, 0, 0, 0, 0, 0, 0, 0, 0, 0, 0, 0, 0, 0, 0, 0, 0, 0, 0, 0, 0, 0, 0, 0, 0, 0, 0, 0, 0, 0, 0, 0, 0, 0, 0, 0, 0, 0, 0, 0, 0, 0, 0, 0, 0, 0, 0, 0, 0, 0, 0, 0, 0, 0, 0, 0, 0, 0, 0, 0, 0, 0, 0, 0, 0, 0, 0, 0, 0, 0, 0, 0, 0, 0, 0, 0, 0, 0, 0, 0, 0, 0, 0, 0, 0, 0, 0, 0, 0, 0, 0, 0, 0, 0, 0, 0, 0, 0, 0, 0, 0, 0]"
    global z_offset_2=[0, 0, 0, 0, 0, 0, 0, 0, 0, 0, 0, 0, 0, 0, 0, 0, 0, 0, 0, 0, 0, 0, 0, 0, 0, 0, 0, 0, 0, 0, 0, 0, 0, 0, 0, 0, 0, 0, 0, 0, 0, 0, 0, 0, 0, 0, 0, 0, 0, 0, 0, 0, 0, 0, 0, 0, 0, 0, 0, 0, 0, 0, 0, 0, 0, 0, 0, 0, 0, 0, 0, 0, 0, 0, 0, 0, 0, 0, 0, 0, 0, 0, 0, 0, 0, 0, 0, 0, 0, 0, 0, 0, 0, 0, 0, 0, 0, 0, 0, 0, 0, 0, 0, 0, 0, 0, 0, 0, 0, 0, 0, 0, 0, 0, 0, 0, 0, 0, 0, 0, 0, 0, 0, 0, 0, 0, 0, 0, 0, 0, 0, 0, 0, 0, 0, 0, 0, 0, 0, 0, 0, 0, 0, 0, 0, 0, 0, 0, 0, 0, 0, 0, 0, 0, 0, 0, 0, 0, 0, 0, 0, 0, 0, 0, 0, 0, 0, 0, 0, 0, 0, 0, 0, 0, 0, 0, 0, 0, 0, 0, 0, 0, 0, 0, 0, 0, 0, 0, 0, 0, 0, 0, 0, 0, 0, 0, 0, 0, 0, 0, 0, 0, 0, 0, 0, 0, 0, 0, 0, 0, 0, 0, 0, 0, 0, 0, 0, 0, 0, 0, 0, 0, 0, 0, 0, 0, 0, 0, 0, 0, 0, 0, 0, 0, 0, 0, 0, 0, 0, 0, 0, 0, 0, 0, 0, 0, 0, 0, 0, 0, 0, 0, 0, 0, 0, 0, 0, 0, 0, 0, 0, 0, 0, 0, 0, 0, 0, 0, 0, 0, 0, 0, 0, 0, 0, 0, 0, 0, 0]
    $ 1618 "z_offset_3≔[0, 0, 0, 0, 0, 0, 0, 0, 0, 0, 0, 0, 0, 0, 0, 0, 0, 0, 0, 0, 0, 0, 0, 0, 0, 0, 0, 0, 0, 0, 0, 0, 0, 0, 0, 0, 0, 0, 0, 0, 0, 0, 0, 0, 0, 0, 0, 0, 0, 0, 0, 0, 0, 0, 0, 0, 0, 0, 0, 0, 0, 0, 0, 0, 0, 0, 0, 0, 0, 0, 0, 0, 0, 0, 0, 0, 0, 0, 0, 0, 0, 0, 0, 0, 0, 0, 0, 0, 0, 0, 0, 0, 0, 0, 0, 0, 0, 0, 0, 0, 0, 0, 0, 0, 0, 0, 0, 0, 0, 0, 0, 0, 0, 0, 0, 0, 0, 0, 0, 0, 0, 0, 0, 0, 0, 0, 0, 0, 0, 0, 0, 0, 0, 0, 0, 0, 0, 0, 0, 0, 0, 0, 0, 0, 0, 0, 0, 0, 0, 0, 0, 0, 0, 0, 0, 0, 0, 0, 0, 0, 0, 0, 0, 0, 0, 0, 0, 0, 0, 0, 0, 0, 0, 0, 0, 0, 0, 0, 0, 0, 0, 0, 0, 0, 0, 0, 0, 0, 0, 0, 0, 0, 0, 0, 0, 0, 0, 0, 0, 0, 0, 0, 0, 0, 0, 0, 0, 0, 0, 0, 0, 0, 0, 0, 0, 0, 0, 0, 0, 0, 0, 0, 0, 0, 0, 0, 0, 0, 0, 0, 0, 0, 0, 0, 0, 0, 0, 0, 0, 0, 0, 0, 0, 0, 0, 0, 0, 0, 0, 0, 0, 0, 0, 0, 0, 0, 0, 0, 0, 0, 0, 0, 0, 0, 0, 0, 0, 0, 0, 0, 0, 0, 0, 0, 0, 0, 0, 0, 0]"
    global z_offset_3=[0, 0, 0, 0, 0, 0, 0, 0, 0, 0, 0, 0, 0, 0, 0, 0, 0, 0, 0, 0, 0, 0, 0, 0, 0, 0, 0, 0, 0, 0, 0, 0, 0, 0, 0, 0, 0, 0, 0, 0, 0, 0, 0, 0, 0, 0, 0, 0, 0, 0, 0, 0, 0, 0, 0, 0, 0, 0, 0, 0, 0, 0, 0, 0, 0, 0, 0, 0, 0, 0, 0, 0, 0, 0, 0, 0, 0, 0, 0, 0, 0, 0, 0, 0, 0, 0, 0, 0, 0, 0, 0, 0, 0, 0, 0, 0, 0, 0, 0, 0, 0, 0, 0, 0, 0, 0, 0, 0, 0, 0, 0, 0, 0, 0, 0, 0, 0, 0, 0, 0, 0, 0, 0, 0, 0, 0, 0, 0, 0, 0, 0, 0, 0, 0, 0, 0, 0, 0, 0, 0, 0, 0, 0, 0, 0, 0, 0, 0, 0, 0, 0, 0, 0, 0, 0, 0, 0, 0, 0, 0, 0, 0, 0, 0, 0, 0, 0, 0, 0, 0, 0, 0, 0, 0, 0, 0, 0, 0, 0, 0, 0, 0, 0, 0, 0, 0, 0, 0, 0, 0, 0, 0, 0, 0, 0, 0, 0, 0, 0, 0, 0, 0, 0, 0, 0, 0, 0, 0, 0, 0, 0, 0, 0, 0, 0, 0, 0, 0, 0, 0, 0, 0, 0, 0, 0, 0, 0, 0, 0, 0, 0, 0, 0, 0, 0, 0, 0, 0, 0, 0, 0, 0, 0, 0, 0, 0, 0, 0, 0, 0, 0, 0, 0, 0, 0, 0, 0, 0, 0, 0, 0, 0, 0, 0, 0, 0, 0, 0, 0, 0, 0, 0, 0, 0, 0, 0, 0, 0, 0]
  end
  def welding_parameter_init():
    $ 1619 "welding_parameter_init" "noBreak"
    $ 1620 "init"
    $ 1621 "If A_sel_v≟A_VL1 or A_sel_v≟A_VL2 or A_sel_v≟A_VR1 or A_sel_v≟A_VR2"
    if (A_sel_v == A_VL1  or  A_sel_v == A_VL2  or  A_sel_v == A_VR1  or  A_sel_v == A_VR2):
      $ 1622 "position_3f2f≔position_3F"
      global position_3f2f=position_3F
      $ 1623 "write_port_register(cell_3f_2f_151,A_sel_v)"
      write_port_register(cell_3f_2f_151,A_sel_v)
      $ 1624 "b8_wv_2f≔ False "
      global b8_wv_2f=  False
      $ 1625 "d_lean_degree≔0"
      global d_lean_degree=0
    else:
      $ 1626 "Else" "noBreak"
      $ 1627 "position_3f2f≔position_2F"
      global position_3f2f=position_2F
      $ 1628 "b8_wv_2f≔ True "
      global b8_wv_2f=  True
      $ 1629 "d_lean_degree≔30"
      global d_lean_degree=30
      $ 1630 "write_port_register(cell_3f_2f_151,A_HOR)"
      write_port_register(cell_3f_2f_151,A_HOR)
    end
    $ 1631 "If current_path≥2"
    if (current_path >= 2):
      $ 1632 "write_port_register(cell_info_152,current_path)"
      write_port_register(cell_info_152,current_path)
    else:
      $ 1633 "Else" "noBreak"
      $ 1634 "write_port_register(cell_info_152,1)"
      write_port_register(cell_info_152,1)
    end
    $ 1635 "write_port_register(return_done_240,0)"
    write_port_register(return_done_240,0)
    $ 1636 "Wait: 0.3"
    sleep(0.3)
    $ 1637 "write_port_register(weld_req_153,1)"
    write_port_register(weld_req_153,1)
    $ 1638 "Wait read_port_register(return_done_240)≟1"
    while (not( read_port_register (return_done_240) == 1)):
      sync()
    end
    $ 1639 "write_port_register(weld_req_153,0)"
    write_port_register(weld_req_153,0)
    $ 1640 "touch_m_check≔0"
    global touch_m_check=0
    $ 1641 "start_end_from_pendant"
    $ 1642 "d_start_current≔read_port_register(244)/10"
    global d_start_current= read_port_register (244)/10
    $ 1643 "d_start_voltage≔read_port_register(245)/10"
    global d_start_voltage= read_port_register (245)/10
    $ 1644 "d_start_time≔read_port_register(241)/10"
    global d_start_time= read_port_register (241)/10
    $ 1645 "d_end_current≔read_port_register(249)/10"
    global d_end_current= read_port_register (249)/10
    $ 1646 "d_end_voltage≔read_port_register(250)/10"
    global d_end_voltage= read_port_register (250)/10
    $ 1647 "d_end_time≔read_port_register(246)/10"
    global d_end_time= read_port_register (246)/10
    $ 1648 "d_end_current_2≔read_port_register(254)/10"
    global d_end_current_2= read_port_register (254)/10
    $ 1649 "d_end_voltage_2≔read_port_register(255)/10"
    global d_end_voltage_2= read_port_register (255)/10
    $ 1650 "d_end_time_2≔read_port_register(251)/10"
    global d_end_time_2= read_port_register (251)/10
    $ 1651 "a7_weld_crater≔[d_start_current,d_start_voltage,d_start_time,d_end_current,d_end_voltage,d_end_time,d_lean_degree]"
    global a7_weld_crater=[d_start_current,d_start_voltage,d_start_time,d_end_current,d_end_voltage,d_end_time,d_lean_degree]
    $ 1652 "a0_volt_ref≔read_port_register(231)/10"
    global a0_volt_ref= read_port_register (231)/10
    $ 1653 "a1_amp_ref≔read_port_register(232)/10"
    global a1_amp_ref= read_port_register (232)/10
    $ 1654 "a2_speed_cpm≔read_port_register(233)/10"
    global a2_speed_cpm= read_port_register (233)/10
    $ 1655 "a3_wv_amplitude≔read_port_register(234)/10"
    global a3_wv_amplitude= read_port_register (234)/10
    $ 1656 "a4_wv_frequency≔read_port_register(225)/10"
    global a4_wv_frequency= read_port_register (225)/10
    $ 1657 "b1_appro_param≔0"
    global b1_appro_param=0
    $ 1658 "b4_wv_delay2≔read_port_register(226)/10"
    global b4_wv_delay2= read_port_register (226)/10
    $ 1659 "b6_wv_delay4≔read_port_register(227)/10"
    global b6_wv_delay4= read_port_register (227)/10
    $ 1660 "'down'"
    # 'down'
    $ 1662 "'up'"
    # 'up'
    $ 1666 "b3_wv_delay1≔0"
    global b3_wv_delay1=0
    $ 1667 "b5_wv_delay3≔0"
    global b5_wv_delay3=0
    $ 1668 "b3_dealy_all≔[b3_wv_delay1,b4_wv_delay2,b5_wv_delay3,b6_wv_delay4]"
    global b3_dealy_all=[b3_wv_delay1,b4_wv_delay2,b5_wv_delay3,b6_wv_delay4]
    $ 1669 "get_width_182≔read_port_register(182)"
    global get_width_182= read_port_register (182)
    $ 1670 "b9_touch_sens≔20"
    global b9_touch_sens=20
    $ 1671 "task_angle≔register_read(228)/10"
    global task_angle=register_read(228)/10
    $ 1672 "Circle_Speed≔a2_speed_cpm"
    global Circle_Speed=a2_speed_cpm
    $ 1673 "CELL_BOTTOM≔a7_cell_bottom"
    global CELL_BOTTOM=a7_cell_bottom
    $ 1674 "a6_scallup_left≔read_port_register(176)"
    global a6_scallup_left= read_port_register (176)
    $ 1675 "a6_scallup_righ≔read_port_register(177)"
    global a6_scallup_righ= read_port_register (177)
    $ 1676 "a5_f_hole≔[a7_cell_bottom,a6_scallup_left,a6_scallup_righ]"
    global a5_f_hole=[a7_cell_bottom,a6_scallup_left,a6_scallup_righ]
    $ 1677 "c8_arc_cur_offs≔read_port_register(239)"
    global c8_arc_cur_offs= read_port_register (239)
    $ 1711 "폴더"
    $ 1712 "offset_2f_x≔7"
    global offset_2f_x=7
    $ 1713 "offset_3f_z≔-5"
    global offset_3f_z=-5
    $ 1714 "If A_sel_v≟A_VR1 or A_sel_v≟A_VR2"
    if (A_sel_v == A_VR1  or  A_sel_v == A_VR2):
      $ 1715 "'3F'"
      # '3F'
      $ 1716 "b2_left_par≔ False "
      global b2_left_par=  False
      $ 1717 "b8_wv_type≔1"
      global b8_wv_type=1
      $ 1718 "If A_sel_v≟A_VR2 and (b1_cell_info_R≟c or b1_cell_info_R≟d)"
      if (A_sel_v == A_VR2  and  (b1_cell_info_R == c  or  b1_cell_info_R == d)):
        $ 1719 "b7_tilt_degree≔[0,0,0]"
        global b7_tilt_degree=[0,0,0]
      else:
        $ 1720 "Else" "noBreak"
        $ 1721 "b7_tilt_degree≔[task_angle,-27,0]"
        global b7_tilt_degree=[task_angle,-27,0]
      end
      $ 1722 "c3_arc_enable≔1"
      global c3_arc_enable=1
    else:
      $ 1723 "ElseIf A_sel_v≟A_VL1 or A_sel_v≟A_VL2"
      if (A_sel_v == A_VL1  or  A_sel_v == A_VL2):
        $ 1724 "'3F'"
        # '3F'
        $ 1725 "b2_left_par≔ True "
        global b2_left_par=  True
        $ 1726 "b8_wv_type≔1"
        global b8_wv_type=1
        $ 1727 "If A_sel_v≟A_VL2 and (b1_cell_info_L≟c or b1_cell_info_L≟d)"
        if (A_sel_v == A_VL2  and  (b1_cell_info_L == c  or  b1_cell_info_L == d)):
          $ 1728 "b7_tilt_degree≔[0,0,0]"
          global b7_tilt_degree=[0,0,0]
        else:
          $ 1729 "Else" "noBreak"
          $ 1730 "b7_tilt_degree≔[task_angle,-27,0]"
          global b7_tilt_degree=[task_angle,-27,0]
        end
        $ 1731 "c3_arc_enable≔1"
        global c3_arc_enable=1
      else:
        $ 1732 "Else" "noBreak"
        $ 1733 "b2_left_par≔ True "
        global b2_left_par=  True
        $ 1734 "b8_wv_type≔2"
        global b8_wv_type=2
        $ 1735 "If A_sel_v≟A_HOR"
        if (A_sel_v == A_HOR):
          $ 1736 "b7_tilt_degree≔[30,-1*task_angle,0]"
          global b7_tilt_degree=[30,-1*task_angle,0]
        else:
          $ 1737 "Else" "noBreak"
          $ 1739 "b7_tilt_degree≔[30,-1*task_angle,0]"
          global b7_tilt_degree=[30,-1*task_angle,0]
        end
        $ 1741 "c3_arc_enable≔1"
        global c3_arc_enable=1
      end
    end
    $ 1742 "If A_sel_v≟A_VL2 or A_sel_v≟A_VR2"
    if (A_sel_v == A_VL2  or  A_sel_v == A_VR2):
      $ 1743 "If b1_cell_info_L≟E or b1_cell_info_L≟e or b1_cell_info_R≟E or b1_cell_info_R≟e"
      if (b1_cell_info_L == E  or  b1_cell_info_L == e  or  b1_cell_info_R == E  or  b1_cell_info_R == e):
        $ 1744 "a8_wv_distance≔read_port_register(182)-a5_f_hole[1]-offset_3f_begin"
        global a8_wv_distance= read_port_register (182)-a5_f_hole[1]-offset_3f_begin
      else:
        $ 1745 "Else" "noBreak"
        $ 1746 "a8_wv_distance≔read_port_register(182)-offset_3f_begin"
        global a8_wv_distance= read_port_register (182)-offset_3f_begin
      end
    else:
      $ 1751 "Else" "noBreak"
      $ 1752 "If b2_left_par"
      if (b2_left_par):
        $ 1753 "Comment"
        # Comment
        $ 1754 "a8_wv_distance≔a6_f_height_l-a5_f_hole[1]-offset_3f_begin"
        global a8_wv_distance=a6_f_height_l-a5_f_hole[1]-offset_3f_begin
        $ 1755 "Comment"
        # Comment
      else:
        $ 1756 "Else" "noBreak"
        $ 1757 "a8_wv_distance≔a6_f_height_r-a5_f_hole[1]-offset_3f_begin"
        global a8_wv_distance=a6_f_height_r-a5_f_hole[1]-offset_3f_begin
      end
    end
    $ 1758 "Ext fun & Squash"
    $ 1759 "If (A_sel_v≟A_VL1 or A_sel_v≟A_VL2) and (b1_cell_info_L≟B or b1_cell_info_L≟D)"
    if ((A_sel_v == A_VL1  or  A_sel_v == A_VL2)  and  (b1_cell_info_L == B  or  b1_cell_info_L == D)):
      $ 1760 "Scallup_check≔ True "
      global Scallup_check=  True
    else:
      $ 1761 "ElseIf (A_sel_v≟A_VR1 or A_sel_v≟A_VR2) and (b1_cell_info_R≟B or b1_cell_info_R≟D)"
      if ((A_sel_v == A_VR1  or  A_sel_v == A_VR2)  and  (b1_cell_info_R == B  or  b1_cell_info_R == D)):
        $ 1762 "Scallup_check≔ True "
        global Scallup_check=  True
      else:
        $ 1763 "Else" "noBreak"
        $ 1764 "Scallup_check≔ False "
        global Scallup_check=  False
      end
    end
    $ 1765 "'squash'"
    # 'squash'
    $ 1766 "If (EXT_flag1[7]≟ True ) and (A_sel_v≠A_HOR) and (A_sel_v≠A_VL2) and (A_sel_v≠A_VR2) and (Scallup_check≟ False ) and (A_sel_v≟A_VL1 and b1_cell_info_L≠E and b1_cell_info_L≠e) and (A_sel_v≟A_VR1 and b1_cell_info_R≠E and b1_cell_info_R≠e)"
    if ((EXT_flag1[7] ==   True  )  and  (A_sel_v != A_HOR)  and  (A_sel_v != A_VL2)  and  (A_sel_v != A_VR2)  and  (Scallup_check ==   False  )  and  (A_sel_v == A_VL1  and  b1_cell_info_L != E  and  b1_cell_info_L != e)  and  (A_sel_v == A_VR1  and  b1_cell_info_R != E  and  b1_cell_info_R != e)):
      $ 1767 "squash"
      $ 1768 "squash_enable≔1"
      global squash_enable=1
      $ 1769 "squash_voltage≔24.5"
      global squash_voltage=24.5
      $ 1770 "squash_current≔190"
      global squash_current=190
      $ 1771 "squash_amp≔7"
      global squash_amp=7
      $ 1772 "squash_speed≔10"
      global squash_speed=10
      $ 1773 "squash_cycle≔8"
      global squash_cycle=8
    else:
      $ 1774 "Else" "noBreak"
      $ 1775 "squash"
      $ 1776 "squash_enable≔0"
      global squash_enable=0
      $ 1777 "squash_voltage≔0"
      global squash_voltage=0
      $ 1778 "squash_current≔0"
      global squash_current=0
      $ 1779 "squash_amp≔0"
      global squash_amp=0
      $ 1780 "squash_speed≔0"
      global squash_speed=0
      $ 1781 "squash_cycle≔0"
      global squash_cycle=0
    end
    $ 1782 "'sladge'"
    # 'sladge'
    $ 1783 "If EXT_flag1[8]≟ True  and EXT_flag1[9]≟ False "
    if (EXT_flag1[8] ==   True    and  EXT_flag1[9] ==   False  ):
      $ 1784 "sludge≔1"
      global sludge=1
    else:
      $ 1785 "ElseIf EXT_flag1[8]≟ False  and EXT_flag1[9]≟ True "
      if (EXT_flag1[8] ==   False    and  EXT_flag1[9] ==   True  ):
        $ 1786 "sludge≔2"
        global sludge=2
      else:
        $ 1787 "Else" "noBreak"
        $ 1788 "sludge≔0"
        global sludge=0
      end
    end
    $ 1789 "waste_cycle≔1"
    global waste_cycle=1
    $ 1790 "c0_offset_x≔read_port_register(229)/10"
    global c0_offset_x= read_port_register (229)/10
    $ 1791 "c0_offset_z≔read_port_register(230)/10"
    global c0_offset_z= read_port_register (230)/10
    $ 1792 "squash_l≔[a0_volt_ref,a1_amp_ref,squash_enable,squash_voltage,squash_current,squash_amp,squash_speed,squash_cycle,waste_cycle,c0_offset_x,c0_offset_z]"
    global squash_l=[a0_volt_ref,a1_amp_ref,squash_enable,squash_voltage,squash_current,squash_amp,squash_speed,squash_cycle,waste_cycle,c0_offset_x,c0_offset_z]
    $ 1793 "WV_gap"
    $ 1794 "c5_wv_gap_y≔read_port_register(236)/10"
    global c5_wv_gap_y= read_port_register (236)/10
    $ 1795 "c6_wv_gap_cpm≔read_port_register(235)/10"
    global c6_wv_gap_cpm= read_port_register (235)/10
    $ 1796 "c9_wv_gap_freq≔a4_wv_frequency"
    global c9_wv_gap_freq=a4_wv_frequency
    $ 1797 "If c6_wv_gap_cpm≟a2_speed_cpm and a3_wv_amplitude≟c5_wv_gap_y"
    if (c6_wv_gap_cpm == a2_speed_cpm  and  a3_wv_amplitude == c5_wv_gap_y):
      $ 1798 "c4_gap_enable≔0"
      global c4_gap_enable=0
    else:
      $ 1799 "Else" "noBreak"
      $ 1800 "c4_gap_enable≔1"
      global c4_gap_enable=1
    end
    $ 1801 "c7_wv_gap≔[c4_gap_enable,c5_wv_gap_y,c6_wv_gap_cpm,c9_wv_gap_freq]"
    global c7_wv_gap=[c4_gap_enable,c5_wv_gap_y,c6_wv_gap_cpm,c9_wv_gap_freq]
    $ 1802 "arc_sen"
    $ 1803 "c3_X_p_gain≔read_port_register(186)/10"
    global c3_X_p_gain= read_port_register (186)/10
    $ 1804 "c3_X_i_gain≔read_port_register(187)/10"
    global c3_X_i_gain= read_port_register (187)/10
    $ 1805 "c3_Z_p_gain≔read_port_register(184)/10"
    global c3_Z_p_gain= read_port_register (184)/10
    $ 1806 "c3_Z_i_gain≔read_port_register(185)/10"
    global c3_Z_i_gain= read_port_register (185)/10
    $ 1807 "c3_wv_arc_fix≔0"
    global c3_wv_arc_fix=0
    $ 1808 "c3_wv_arc≔[c3_arc_enable,c3_X_p_gain,c3_X_i_gain,c3_Z_p_gain,c3_Z_i_gain,c3_wv_arc_fix]"
    global c3_wv_arc=[c3_arc_enable,c3_X_p_gain,c3_X_i_gain,c3_Z_p_gain,c3_Z_i_gain,c3_wv_arc_fix]
    $ 1809 "volt and current"
    $ 1810 "set_current_voltage(a1_amp_ref,a0_volt_ref)"
    set_current_voltage(a1_amp_ref,a0_volt_ref)
    $ 1811 "write_port_register(154,1)"
    write_port_register(154,1)
    $ 1812 "Wait read_port_register(return_done_240)≟0"
    while (not( read_port_register (return_done_240) == 0)):
      sync()
    end
    $ 1813 "write_port_register(154,0)"
    write_port_register(154,0)
  end
  def welding_parameter_sim():
    $ 1814 "welding_parameter_sim" "noBreak"
    $ 1815 "init"
    $ 1816 "If A_sel_v≟A_VL1 or A_sel_v≟A_VL2 or A_sel_v≟A_VR1 or A_sel_v≟A_VR2"
    if (A_sel_v == A_VL1  or  A_sel_v == A_VL2  or  A_sel_v == A_VR1  or  A_sel_v == A_VR2):
      $ 1817 "position_3f2f≔position_3F"
      global position_3f2f=position_3F
      $ 1818 "write_port_register(cell_3f_2f_151,A_sel_v)"
      write_port_register(cell_3f_2f_151,A_sel_v)
      $ 1819 "b8_wv_2f≔ False "
      global b8_wv_2f=  False
      $ 1820 "d_lean_degree≔0"
      global d_lean_degree=0
    else:
      $ 1821 "Else" "noBreak"
      $ 1822 "position_3f2f≔position_2F"
      global position_3f2f=position_2F
      $ 1823 "b8_wv_2f≔ True "
      global b8_wv_2f=  True
      $ 1824 "d_lean_degree≔30"
      global d_lean_degree=30
      $ 1825 "write_port_register(cell_3f_2f_151,A_HOR)"
      write_port_register(cell_3f_2f_151,A_HOR)
    end
    $ 1826 "If current_path≥2"
    if (current_path >= 2):
      $ 1827 "write_port_register(cell_info_152,current_path)"
      write_port_register(cell_info_152,current_path)
    else:
      $ 1828 "Else" "noBreak"
      $ 1829 "write_port_register(cell_info_152,1)"
      write_port_register(cell_info_152,1)
    end
    $ 1830 "write_port_register(return_done_240,0)"
    write_port_register(return_done_240,0)
    $ 1831 "Wait: 0.3"
    sleep(0.3)
    $ 1832 "write_port_register(weld_req_153,1)"
    write_port_register(weld_req_153,1)
    $ 1834 "write_port_register(weld_req_153,0)"
    write_port_register(weld_req_153,0)
    $ 1835 "touch_m_check≔0"
    global touch_m_check=0
    $ 1836 "start_end_from_pendant"
    $ 1837 "d_start_current≔read_port_register(244)/10"
    global d_start_current= read_port_register (244)/10
    $ 1838 "d_start_voltage≔read_port_register(245)/10"
    global d_start_voltage= read_port_register (245)/10
    $ 1839 "d_start_time≔read_port_register(241)/10"
    global d_start_time= read_port_register (241)/10
    $ 1840 "d_end_current≔read_port_register(249)/10"
    global d_end_current= read_port_register (249)/10
    $ 1841 "d_end_voltage≔read_port_register(250)/10"
    global d_end_voltage= read_port_register (250)/10
    $ 1842 "d_end_time≔read_port_register(246)/10"
    global d_end_time= read_port_register (246)/10
    $ 1843 "d_end_current_2≔read_port_register(254)/10"
    global d_end_current_2= read_port_register (254)/10
    $ 1844 "d_end_voltage_2≔read_port_register(255)/10"
    global d_end_voltage_2= read_port_register (255)/10
    $ 1845 "d_end_time_2≔read_port_register(251)/10"
    global d_end_time_2= read_port_register (251)/10
    $ 1846 "a7_weld_crater≔[d_start_current,d_start_voltage,d_start_time,d_end_current,d_end_voltage,d_end_time,d_lean_degree]"
    global a7_weld_crater=[d_start_current,d_start_voltage,d_start_time,d_end_current,d_end_voltage,d_end_time,d_lean_degree]
    $ 1847 "a0_volt_ref≔read_port_register(231)/10"
    global a0_volt_ref= read_port_register (231)/10
    $ 1848 "a1_amp_ref≔read_port_register(232)/10"
    global a1_amp_ref= read_port_register (232)/10
    $ 1849 "b1_appro_param≔0"
    global b1_appro_param=0
    $ 1850 "Folder"
    $ 1851 "a2_speed_cpm≔17"
    global a2_speed_cpm=17
    $ 1852 "a3_wv_amplitude≔5"
    global a3_wv_amplitude=5
    $ 1853 "a4_wv_frequency≔1.4"
    global a4_wv_frequency=1.4
    $ 1854 "b4_wv_delay2≔0.3"
    global b4_wv_delay2=0.3
    $ 1855 "b6_wv_delay4≔0.3"
    global b6_wv_delay4=0.3
    $ 1856 "b9_touch_sens≔10"
    global b9_touch_sens=10
    $ 1857 "task_angle≔0"
    global task_angle=0
    $ 1858 "a6_scallup_left≔0"
    global a6_scallup_left=0
    $ 1859 "a6_scallup_righ≔0"
    global a6_scallup_righ=0
    $ 1860 "b3_wv_delay1≔0"
    global b3_wv_delay1=0
    $ 1861 "b5_wv_delay3≔0"
    global b5_wv_delay3=0
    $ 1862 "b3_dealy_all≔[b3_wv_delay1,b4_wv_delay2,b5_wv_delay3,b6_wv_delay4]"
    global b3_dealy_all=[b3_wv_delay1,b4_wv_delay2,b5_wv_delay3,b6_wv_delay4]
    $ 1863 "get_width_182≔a6_callar_vert"
    global get_width_182=a6_callar_vert
    $ 1864 "task_angle≔register_read(228)/10"
    global task_angle=register_read(228)/10
    $ 1865 "Circle_Speed≔a2_speed_cpm"
    global Circle_Speed=a2_speed_cpm
    $ 1866 "CELL_BOTTOM≔a7_cell_bottom"
    global CELL_BOTTOM=a7_cell_bottom
    $ 1867 "a5_f_hole≔[a7_cell_bottom,a6_scallup_left,a6_scallup_righ]"
    global a5_f_hole=[a7_cell_bottom,a6_scallup_left,a6_scallup_righ]
    $ 1868 "폴더"
    $ 1869 "offset_2f_x≔7"
    global offset_2f_x=7
    $ 1870 "offset_3f_z≔-5"
    global offset_3f_z=-5
    $ 1871 "If A_sel_v≟A_VR1 or A_sel_v≟A_VR2"
    if (A_sel_v == A_VR1  or  A_sel_v == A_VR2):
      $ 1872 "'3F'"
      # '3F'
      $ 1873 "b2_left_par≔ False "
      global b2_left_par=  False
      $ 1874 "b8_wv_type≔1"
      global b8_wv_type=1
      $ 1875 "b7_tilt_degree≔[task_angle,-27,0]"
      global b7_tilt_degree=[task_angle,-27,0]
      $ 1876 "c3_arc_enable≔1"
      global c3_arc_enable=1
    else:
      $ 1877 "ElseIf A_sel_v≟A_VL1 or A_sel_v≟A_VL2"
      if (A_sel_v == A_VL1  or  A_sel_v == A_VL2):
        $ 1878 "'3F'"
        # '3F'
        $ 1879 "b2_left_par≔ True "
        global b2_left_par=  True
        $ 1880 "b8_wv_type≔1"
        global b8_wv_type=1
        $ 1881 "b7_tilt_degree≔[task_angle,-27,0]"
        global b7_tilt_degree=[task_angle,-27,0]
        $ 1882 "c3_arc_enable≔1"
        global c3_arc_enable=1
      else:
        $ 1883 "Else" "noBreak"
        $ 1884 "b2_left_par≔ True "
        global b2_left_par=  True
        $ 1885 "b8_wv_type≔2"
        global b8_wv_type=2
        $ 1886 "b7_tilt_degree≔[30,-1*task_angle,0]"
        global b7_tilt_degree=[30,-1*task_angle,0]
        $ 1888 "c3_arc_enable≔0"
        global c3_arc_enable=0
      end
    end
    $ 1889 "If A_sel_v≟A_VL2 or A_sel_v≟A_VR2"
    if (A_sel_v == A_VL2  or  A_sel_v == A_VR2):
      $ 1890 "a8_wv_distance≔read_port_register(182)"
      global a8_wv_distance= read_port_register (182)
    else:
      $ 1895 "Else" "noBreak"
      $ 1896 "If b2_left_par"
      if (b2_left_par):
        $ 1897 "Comment"
        # Comment
        $ 1898 "a8_wv_distance≔a6_f_height_l-a5_f_hole[1]"
        global a8_wv_distance=a6_f_height_l-a5_f_hole[1]
        $ 1899 "Comment"
        # Comment
      else:
        $ 1900 "Else" "noBreak"
        $ 1901 "a8_wv_distance≔a6_f_height_r-a5_f_hole[1]"
        global a8_wv_distance=a6_f_height_r-a5_f_hole[1]
      end
    end
    $ 1902 "Ext fun & Squash"
    $ 1903 "If (A_sel_v≟A_VL1 or A_sel_v≟A_VL2) and (b1_cell_info_L≟B or b1_cell_info_L≟D)"
    if ((A_sel_v == A_VL1  or  A_sel_v == A_VL2)  and  (b1_cell_info_L == B  or  b1_cell_info_L == D)):
      $ 1904 "Scallup_check≔ True "
      global Scallup_check=  True
    else:
      $ 1905 "ElseIf (A_sel_v≟A_VR1 or A_sel_v≟A_VR2) and (b1_cell_info_R≟B or b1_cell_info_R≟D)"
      if ((A_sel_v == A_VR1  or  A_sel_v == A_VR2)  and  (b1_cell_info_R == B  or  b1_cell_info_R == D)):
        $ 1906 "Scallup_check≔ True "
        global Scallup_check=  True
      else:
        $ 1907 "Else" "noBreak"
        $ 1908 "Scallup_check≔ False "
        global Scallup_check=  False
      end
    end
    $ 1909 "If (EXT_flag1[7]≟ True ) and (A_sel_v≠A_HOR) and (A_sel_v≠A_VL2) and (A_sel_v≠A_VR2) and (Scallup_check≟ False )"
    if ((EXT_flag1[7] ==   True  )  and  (A_sel_v != A_HOR)  and  (A_sel_v != A_VL2)  and  (A_sel_v != A_VR2)  and  (Scallup_check ==   False  )):
      $ 1910 "squash"
      $ 1911 "squash_enable≔1"
      global squash_enable=1
      $ 1912 "squash_voltage≔24.5"
      global squash_voltage=24.5
      $ 1913 "squash_current≔190"
      global squash_current=190
      $ 1914 "squash_amp≔7"
      global squash_amp=7
      $ 1915 "squash_speed≔10"
      global squash_speed=10
      $ 1916 "squash_cycle≔8"
      global squash_cycle=8
    else:
      $ 1917 "Else" "noBreak"
      $ 1918 "squash"
      $ 1919 "squash_enable≔0"
      global squash_enable=0
      $ 1920 "squash_voltage≔0"
      global squash_voltage=0
      $ 1921 "squash_current≔0"
      global squash_current=0
      $ 1922 "squash_amp≔0"
      global squash_amp=0
      $ 1923 "squash_speed≔0"
      global squash_speed=0
      $ 1924 "squash_cycle≔0"
      global squash_cycle=0
    end
    $ 1925 "waste_cycle≔2"
    global waste_cycle=2
    $ 1926 "c0_offset_x≔read_port_register(229)/10"
    global c0_offset_x= read_port_register (229)/10
    $ 1927 "c0_offset_z≔read_port_register(230)/10"
    global c0_offset_z= read_port_register (230)/10
    $ 1928 "squash_l≔[a0_volt_ref,a1_amp_ref,squash_enable,squash_voltage,squash_current,squash_amp,squash_speed,squash_cycle,waste_cycle,c0_offset_x,c0_offset_z]"
    global squash_l=[a0_volt_ref,a1_amp_ref,squash_enable,squash_voltage,squash_current,squash_amp,squash_speed,squash_cycle,waste_cycle,c0_offset_x,c0_offset_z]
    $ 1929 "WV_gap"
    $ 1930 "c5_wv_gap_y≔a3_wv_amplitude"
    global c5_wv_gap_y=a3_wv_amplitude
    $ 1931 "c6_wv_gap_cpm≔a2_speed_cpm"
    global c6_wv_gap_cpm=a2_speed_cpm
    $ 1932 "c9_wv_gap_freq≔a4_wv_frequency"
    global c9_wv_gap_freq=a4_wv_frequency
    $ 1933 "If c6_wv_gap_cpm≟a2_speed_cpm and a3_wv_amplitude≟c5_wv_gap_y"
    if (c6_wv_gap_cpm == a2_speed_cpm  and  a3_wv_amplitude == c5_wv_gap_y):
      $ 1934 "c4_gap_enable≔0"
      global c4_gap_enable=0
    else:
      $ 1935 "Else" "noBreak"
      $ 1936 "c4_gap_enable≔1"
      global c4_gap_enable=1
    end
    $ 1937 "c4_gap_enable≔0"
    global c4_gap_enable=0
    $ 1938 "c7_wv_gap≔[c4_gap_enable,c5_wv_gap_y,c6_wv_gap_cpm,c9_wv_gap_freq]"
    global c7_wv_gap=[c4_gap_enable,c5_wv_gap_y,c6_wv_gap_cpm,c9_wv_gap_freq]
    $ 1939 "arc_sen"
    $ 1940 "c3_X_p_gain≔read_port_register(186)/10"
    global c3_X_p_gain= read_port_register (186)/10
    $ 1941 "c3_X_i_gain≔read_port_register(187)/10"
    global c3_X_i_gain= read_port_register (187)/10
    $ 1942 "c3_Z_p_gain≔read_port_register(184)/10"
    global c3_Z_p_gain= read_port_register (184)/10
    $ 1943 "c3_Z_i_gain≔read_port_register(185)/10"
    global c3_Z_i_gain= read_port_register (185)/10
    $ 1944 "c3_wv_arc_fix≔0"
    global c3_wv_arc_fix=0
    $ 1945 "c3_wv_arc≔[c3_arc_enable,c3_X_p_gain,c3_X_i_gain,c3_Z_p_gain,c3_Z_i_gain,c3_wv_arc_fix]"
    global c3_wv_arc=[c3_arc_enable,c3_X_p_gain,c3_X_i_gain,c3_Z_p_gain,c3_Z_i_gain,c3_wv_arc_fix]
    $ 1946 "volt and current"
    $ 1947 "set_current_voltage(a1_amp_ref,a0_volt_ref)"
    set_current_voltage(a1_amp_ref,a0_volt_ref)
    $ 1948 "write_port_register(154,1)"
    write_port_register(154,1)
    $ 1950 "write_port_register(154,0)"
    write_port_register(154,0)
  end
  def Move_done():
    $ 1951 "Move_done" "noBreak"
    $ 1952 "write_port_register(robot_move_163,0)"
    write_port_register(robot_move_163,0)
    $ 1953 "write_port_register(robot_pose_164,0)"
    write_port_register(robot_pose_164,0)
    $ 1954 "write_port_register(robot_ready_141,1)"
    write_port_register(robot_ready_141,1)
  end
  def MoveFun():
    $ 1955 "MoveFun" "noBreak"
    $ 1956 "b_touch_pos≔A_Prepos_l[A_sel_v]"
    global b_touch_pos=A_Prepos_l[A_sel_v]
    $ 1957 "MoveL"
    $ 1958 "b_touch_pos" "breakAfter"
    movel(pose_trans(Base, b_touch_pos), a=0.35, v=0.35)
  end
  def MoveFun_cd():
    $ 1959 "MoveFun_cd" "noBreak"
    $ 1960 "b_touch_pos≔A_Prepos_l[A_sel_v]"
    global b_touch_pos=A_Prepos_l[A_sel_v]
    $ 1961 "If A_sel_v≟A_VR2 and (b1_cell_info_R≟c or b1_cell_info_R≟d)"
    if (A_sel_v == A_VR2  and  (b1_cell_info_R == c  or  b1_cell_info_R == d)):
      $ 1962 "tilt_deg≔27"
      global tilt_deg=27
      $ 1963 "tilt_deg_ry≔19"
      global tilt_deg_ry=19
      $ 1964 "tilt_deg_rz≔0"
      global tilt_deg_rz=0
    else:
      $ 1965 "Else" "noBreak"
      $ 1966 "tilt_deg≔10"
      global tilt_deg=10
      $ 1967 "tilt_deg_ry≔5"
      global tilt_deg_ry=5
      $ 1968 "tilt_deg_rz≔0"
      global tilt_deg_rz=0
    end
    $ 1969 "If b2_left_par"
    if (b2_left_par):
      $ 1970 "b_touch_pos≔pose_add(b_touch_pos, p[0,18/1000,0,0,0,0])"
      global b_touch_pos= pose_add (b_touch_pos, p[0,18/1000,0,0,0,0])
      $ 1971 "b_touch_pos≔pose_trans(b_touch_pos, p[0,0,0,d2r(-tilt_deg),d2r(-tilt_deg_ry),d2r(tilt_deg_rz)])"
      global b_touch_pos= pose_trans (b_touch_pos, p[0,0,0,d2r(-tilt_deg),d2r(-tilt_deg_ry),d2r(tilt_deg_rz)])
    else:
      $ 1972 "Else" "noBreak"
      $ 1973 "b_touch_pos≔pose_add(b_touch_pos, p[0,-18/1000,0,0,0,0])"
      global b_touch_pos= pose_add (b_touch_pos, p[0,-18/1000,0,0,0,0])
      $ 1974 "b_touch_pos≔pose_trans(b_touch_pos, p[0,0,0,d2r(tilt_deg),d2r(-tilt_deg_ry),d2r(-tilt_deg_rz)])"
      global b_touch_pos= pose_trans (b_touch_pos, p[0,0,0,d2r(tilt_deg),d2r(-tilt_deg_ry),d2r(-tilt_deg_rz)])
    end
    $ 1975 "MoveL"
    $ 1976 "b_touch_pos" "breakAfter"
    movel(pose_trans(Base, b_touch_pos), a=0.35, v=0.35)
  end
  def MoveandTouchFun_2f():
    $ 1977 "MoveandTouchFun_2f" "noBreak"
    $ 1978 "b_touch_pos≔A_Prepos_l[A_sel_v]"
    global b_touch_pos=A_Prepos_l[A_sel_v]
    $ 1979 "tilt_deg≔3"
    global tilt_deg=3
    $ 1980 "tilt_deg_ry≔3"
    global tilt_deg_ry=3
    $ 1981 "tilt_deg_rz≔0"
    global tilt_deg_rz=0
    $ 1982 "If  False "
    if (  False  ):
      $ 1983 "Wait: 0.01"
      sleep(0.01)
    else:
      $ 1984 "ElseIf A_sel_v≟A_HOR and b1_cell_info_L≟E"
      if (A_sel_v == A_HOR  and  b1_cell_info_L == E):
        $ 1985 "tilt_deg≔6"
        global tilt_deg=6
        $ 1986 "tilt_deg_ry≔-5"
        global tilt_deg_ry=-5
        $ 1987 "tilt_deg_rz≔0"
        global tilt_deg_rz=0
        $ 1988 "b_touch_pos≔pose_trans(b_touch_pos, p[0,0/1000,0,d2r(tilt_deg),d2r(-tilt_deg_ry),d2r(tilt_deg_rz)])"
        global b_touch_pos= pose_trans (b_touch_pos, p[0,0/1000,0,d2r(tilt_deg),d2r(-tilt_deg_ry),d2r(tilt_deg_rz)])
      else:
        $ 1989 "ElseIf A_sel_v≟A_HOR_R and b1_cell_info_R≟E"
        if (A_sel_v == A_HOR_R  and  b1_cell_info_R == E):
          $ 1990 "tilt_deg≔6"
          global tilt_deg=6
          $ 1991 "tilt_deg_ry≔-5"
          global tilt_deg_ry=-5
          $ 1992 "tilt_deg_rz≔0"
          global tilt_deg_rz=0
          $ 1993 "b_touch_pos≔pose_trans(b_touch_pos, p[0,0/1000,0,d2r(tilt_deg),d2r(-tilt_deg_ry),d2r(-tilt_deg_rz)])"
          global b_touch_pos= pose_trans (b_touch_pos, p[0,0/1000,0,d2r(tilt_deg),d2r(-tilt_deg_ry),d2r(-tilt_deg_rz)])
        else:
          $ 1994 "ElseIf b2_left_par"
          if (b2_left_par):
            $ 1995 "b_touch_pos≔pose_trans(b_touch_pos, p[0,0/1000,0,d2r(tilt_deg),d2r(-tilt_deg_ry),d2r(tilt_deg_rz)])"
            global b_touch_pos= pose_trans (b_touch_pos, p[0,0/1000,0,d2r(tilt_deg),d2r(-tilt_deg_ry),d2r(tilt_deg_rz)])
          else:
            $ 1996 "Else" "noBreak"
            $ 1997 "b_touch_pos≔pose_trans(b_touch_pos, p[0,0/1000,0,d2r(tilt_deg),d2r(-tilt_deg_ry),d2r(-tilt_deg_rz)])"
            global b_touch_pos= pose_trans (b_touch_pos, p[0,0/1000,0,d2r(tilt_deg),d2r(-tilt_deg_ry),d2r(-tilt_deg_rz)])
          end
        end
      end
    end
    $ 1998 "MoveL"
    $ 1999 "b_touch_pos" "breakAfter"
    movel(pose_trans(Base, b_touch_pos), a=0.35, v=0.35)
    $ 2000 "Touch_2f"
    $ 2001 "If  False "
    if (  False  ):
      $ 2002 "Wait: 0.01"
      sleep(0.01)
    else:
      $ 2003 "ElseIf A_sel_v≟A_HOR and b1_cell_info_L≟E"
      if (A_sel_v == A_HOR  and  b1_cell_info_L == E):
        $ 2004 "tilt_deg≔3"
        global tilt_deg=3
        $ 2005 "tilt_deg_ry≔3"
        global tilt_deg_ry=3
        $ 2006 "tilt_deg_rz≔0"
        global tilt_deg_rz=0
        $ 2007 "b_touch_pos2≔pose_trans(b_touch_pos, p[0,0/1000,0,d2r(tilt_deg),d2r(-tilt_deg_ry),d2r(tilt_deg_rz)])"
        global b_touch_pos2= pose_trans (b_touch_pos, p[0,0/1000,0,d2r(tilt_deg),d2r(-tilt_deg_ry),d2r(tilt_deg_rz)])
        $ 2008 "touch_result≔touch_fun_2f(b_touch_pos,b_touch_pos2,b2_left_par,b9_touch_sens)"
        global touch_result=touch_fun_2f(b_touch_pos,b_touch_pos2,b2_left_par,b9_touch_sens)
      else:
        $ 2009 "ElseIf A_sel_v≟A_HOR_R and b1_cell_info_R≟E"
        if (A_sel_v == A_HOR_R  and  b1_cell_info_R == E):
          $ 2010 "tilt_deg≔3"
          global tilt_deg=3
          $ 2011 "tilt_deg_ry≔3"
          global tilt_deg_ry=3
          $ 2012 "tilt_deg_rz≔0"
          global tilt_deg_rz=0
          $ 2013 "b_touch_pos2≔pose_trans(b_touch_pos, p[0,0/1000,0,d2r(tilt_deg),d2r(-tilt_deg_ry),d2r(-tilt_deg_rz)])"
          global b_touch_pos2= pose_trans (b_touch_pos, p[0,0/1000,0,d2r(tilt_deg),d2r(-tilt_deg_ry),d2r(-tilt_deg_rz)])
          $ 2014 "touch_result≔touch_fun_2f(b_touch_pos,b_touch_pos2,b2_left_par,b9_touch_sens)"
          global touch_result=touch_fun_2f(b_touch_pos,b_touch_pos2,b2_left_par,b9_touch_sens)
        else:
          $ 2015 "Else" "noBreak"
          $ 2016 "touch_result≔touch_fun_2f(b_touch_pos,b_touch_pos,b2_left_par,b9_touch_sens)"
          global touch_result=touch_fun_2f(b_touch_pos,b_touch_pos,b2_left_par,b9_touch_sens)
        end
      end
    end
    $ 2018 "If b2_left_par"
    if (b2_left_par):
      $ 2019 "touch_result≔feature_offset(touch_result,p[0,(Touch_dis)/1000,0,0,0,0],center_line)"
      global touch_result=feature_offset(touch_result,p[0,(Touch_dis)/1000,0,0,0,0],center_line)
    else:
      $ 2021 "Else" "noBreak"
      $ 2022 "touch_result≔feature_offset(touch_result,p[0,(-Touch_dis)/1000,0,0,0,0],center_line)"
      global touch_result=feature_offset(touch_result,p[0,(-Touch_dis)/1000,0,0,0,0],center_line)
    end
    $ 2024 "A_Touch_p[A_sel_v]=touch_result"
    A_Touch_p[A_sel_v]=touch_result
    $ 2025 "If EXT_flag1[3]≟ True "
    if (EXT_flag1[3] ==   True  ):
      $ 2026 "MoveL"
      $ 2027 "manual_tp≔tilt_2f_fun(touch_result,basic_tilt_2f,wv_direction)"
      global manual_tp=tilt_2f_fun(touch_result,basic_tilt_2f,wv_direction)
      $ 2028 "manual_tp≔pose_trans(manual_tp, p[0,0,-10/1000,0,0,0])"
      global manual_tp= pose_trans (manual_tp, p[0,0,-10/1000,0,0,0])
      $ 2029 "manual_tp" "breakAfter"
      movel(pose_trans(Base, manual_tp), a=0.3, v=0.15)
      $ 2030 "Wait: 1.5"
      sleep(1.5)
    end
  end
  def MoveandTouchFun_3f():
    $ 2031 "MoveandTouchFun_3f" "noBreak"
    $ 2032 "b_touch_pos≔A_Prepos_l[A_sel_v]"
    global b_touch_pos=A_Prepos_l[A_sel_v]
    $ 2033 "tilt_deg_ry≔0"
    global tilt_deg_ry=0
    $ 2034 "tilt_deg_rz≔0"
    global tilt_deg_rz=0
    $ 2035 "If b2_left_par"
    if (b2_left_par):
      $ 2036 "tilt_deg≔6"
      global tilt_deg=6
      $ 2037 "b_touch_pos≔pose_trans(b_touch_pos, p[0,0/1000,0,d2r(tilt_deg),d2r(tilt_deg_ry),d2r(tilt_deg_rz)])"
      global b_touch_pos= pose_trans (b_touch_pos, p[0,0/1000,0,d2r(tilt_deg),d2r(tilt_deg_ry),d2r(tilt_deg_rz)])
    else:
      $ 2038 "Else" "noBreak"
      $ 2039 "tilt_deg≔0.5"
      global tilt_deg=0.5
      $ 2040 "b_touch_pos≔pose_trans(b_touch_pos, p[0,0/1000,0,d2r(-tilt_deg),d2r(tilt_deg_ry),d2r(tilt_deg_rz)])"
      global b_touch_pos= pose_trans (b_touch_pos, p[0,0/1000,0,d2r(-tilt_deg),d2r(tilt_deg_ry),d2r(tilt_deg_rz)])
    end
    $ 2051 "move_pre"
    $ 2052 "If (b2_left_par≟ True  and point_dist(A_Prepos_l[A_HOR], A_Prepos_l[A_VL1])>0.032) or (b2_left_par≟ False  and point_dist(A_Prepos_l[A_HOR_R],A_Prepos_l[A_VR1])>0.032)"
    if ((b2_left_par ==   True    and  point_dist(A_Prepos_l[A_HOR], A_Prepos_l[A_VL1])>0.032)  or  (b2_left_par ==   False    and  point_dist(A_Prepos_l[A_HOR_R],A_Prepos_l[A_VR1])>0.032)):
      $ 2053 "if move from home"
      $ 2054 "j_cp≔get_actual_joint_positions()"
      global j_cp= get_actual_joint_positions ()
      $ 2055 "If b2_left_par"
      if (b2_left_par):
        $ 2056 "If norm(b_touch_pos[1]*1000)>300"
        if (norm(b_touch_pos[1]*1000)>300):
          $ 2057 "inner_p≔p[-15/1000,-35/1000,0,0,0,0]"
          global inner_p=p[-15/1000,-35/1000,0,0,0,0]
        else:
          $ 2058 "Else" "noBreak"
          $ 2059 "inner_p≔p[0,0,0,0,0,0]"
          global inner_p=p[0,0,0,0,0,0]
        end
        $ 2060 "j_tp≔get_inverse_kin(pose_add(b_touch_pos,inner_p),qnear=left_j)"
        global j_tp= get_inverse_kin (pose_add(b_touch_pos,inner_p),qnear=left_j)
      else:
        $ 2061 "Else" "noBreak"
        $ 2062 "If norm(b_touch_pos[1]*1000)>300"
        if (norm(b_touch_pos[1]*1000)>300):
          $ 2063 "inner_p≔p[-15/1000,35/1000,0,0,0,0]"
          global inner_p=p[-15/1000,35/1000,0,0,0,0]
        else:
          $ 2064 "Else" "noBreak"
          $ 2065 "inner_p≔p[0,0,0,0,0,0]"
          global inner_p=p[0,0,0,0,0,0]
        end
        $ 2066 "j_tp≔get_inverse_kin(pose_add(b_touch_pos,inner_p),qnear=right_j)"
        global j_tp= get_inverse_kin ( pose_add (b_touch_pos,inner_p),qnear=right_j)
      end
      $ 2067 "j_cp[0]=j_tp[0]"
      j_cp[0]=j_tp[0]
      $ 2068 "j_cp[1]=j_cp[1]+(j_tp[1]-j_cp[1])/2"
      j_cp[1]=j_cp[1]+(j_tp[1]-j_cp[1])/2
      $ 2069 "j_cp[2]=j_cp[2]+(j_tp[2]-j_cp[2])/2.5"
      j_cp[2]=j_cp[2]+(j_tp[2]-j_cp[2])/2.5
      $ 2070 "j_cp[3]=j_cp[3]+(j_tp[3]-j_cp[3])/2.5"
      j_cp[3]=j_cp[3]+(j_tp[3]-j_cp[3])/2.5
      $ 2071 "j_cp[4]=j_cp[4]+(j_tp[4]-j_cp[4])/3"
      j_cp[4]=j_cp[4]+(j_tp[4]-j_cp[4])/3
      $ 2072 "j_cp[5]=j_cp[5]+(j_tp[5]-j_cp[5])/1"
      j_cp[5]=j_cp[5]+(j_tp[5]-j_cp[5])/1
      $ 2073 "MoveJ"
      $ 2074 "j_cp" "breakAfter"
      movej(j_cp, a=1.3962634015954636, v=1.0471975511965976)
      $ 2075 "j_tp≔[j_cp[0],j_cp[1],j_cp[2],j_cp[3],j_tp[4],j_tp[5]]"
      global j_tp=[j_cp[0],j_cp[1],j_cp[2],j_cp[3],j_tp[4],j_tp[5]]
    end
    $ 2078 "MoveL"
    $ 2079 "b_touch_pos" "breakAfter"
    movel(pose_trans(Base, b_touch_pos), a=0.35, v=0.35)
    $ 2082 "touch_3f_down"
    $ 2084 "touch_result≔touch_fun2(b_touch_pos,b2_left_par,b9_touch_sens,b2_par_cd)"
    global touch_result=touch_fun2(b_touch_pos,b2_left_par,b9_touch_sens,b2_par_cd)
    $ 2085 "If Scallup_check≟ False "
    if (Scallup_check ==   False  ):
      $ 2086 "touch_result≔pose_trans(touch_result,p[-(Touch_dis)/1000,0,0,0,0,0])"
      global touch_result= pose_trans (touch_result,p[-(Touch_dis)/1000,0,0,0,0,0])
    else:
      $ 2087 "Else" "noBreak"
      $ 2088 "Scallup_check≔ False "
      global Scallup_check=  False
    end
    $ 2091 "A_Touch_p[A_sel_v]=touch_result"
    A_Touch_p[A_sel_v]=touch_result
    $ 2092 "If EXT_flag1[3]≟ True "
    if (EXT_flag1[3] ==   True  ):
      $ 2093 "MoveL"
      $ 2094 "manual_tp≔tilt_3f_fun(A_Touch_p[A_sel_v],basic_tilt_3f,0)"
      global manual_tp=tilt_3f_fun(A_Touch_p[A_sel_v],basic_tilt_3f,0)
      $ 2095 "manual_tp≔pose_trans(manual_tp, p[0,0,-10/1000,0,0,0])"
      global manual_tp= pose_trans (manual_tp, p[0,0,-10/1000,0,0,0])
      $ 2096 "manual_tp" "breakAfter"
      movel(pose_trans(Base, manual_tp), a=0.3, v=0.15)
      $ 2097 "Wait: 1.5"
      sleep(1.5)
    end
  end
  def weav_welding_3f():
    $ 2117 "weav_welding_3f" "noBreak"
    $ 2118 "If running_trig≟ True "
    global thread_flag_2118=0
    thread Thread_if_2118():
      $ 2119 "inv_inching(inv_inch_time)"
      inv_inching(inv_inch_time)
      $ 2120 "b_touch_pos≔A_Prepos_l[A_sel_v]"
      global b_touch_pos=A_Prepos_l[A_sel_v]
      $ 2121 "move_pre"
      $ 2122 "If (b2_left_par≟ True  and point_dist(A_Prepos_l[A_HOR], A_Prepos_l[A_VL1])>0.032) or (b2_left_par≟ False  and point_dist(A_Prepos_l[A_HOR_R],A_Prepos_l[A_VR1])>0.032)"
      if ((b2_left_par ==   True    and  point_dist(A_Prepos_l[A_HOR], A_Prepos_l[A_VL1])>0.032)  or  (b2_left_par ==   False    and  point_dist(A_Prepos_l[A_HOR_R],A_Prepos_l[A_VR1])>0.032)):
        $ 2123 "if move from home"
        $ 2124 "j_cp≔get_actual_joint_positions()"
        global j_cp= get_actual_joint_positions ()
        $ 2125 "If b2_left_par"
        if (b2_left_par):
          $ 2126 "If norm(b_touch_pos[1]*1000)>300"
          if (norm(b_touch_pos[1]*1000)>300):
            $ 2127 "inner_p≔p[-15/1000,-35/1000,0,0,0,0]"
            global inner_p=p[-15/1000,-35/1000,0,0,0,0]
          else:
            $ 2128 "Else" "noBreak"
            $ 2129 "inner_p≔p[0,0,0,0,0,0]"
            global inner_p=p[0,0,0,0,0,0]
          end
          $ 2130 "j_tp≔get_inverse_kin(pose_add(b_touch_pos,inner_p),qnear=left_j)"
          global j_tp= get_inverse_kin (pose_add(b_touch_pos,inner_p),qnear=left_j)
        else:
          $ 2131 "Else" "noBreak"
          $ 2132 "If norm(b_touch_pos[1]*1000)>300"
          if (norm(b_touch_pos[1]*1000)>300):
            $ 2133 "inner_p≔p[-15/1000,35/1000,0,0,0,0]"
            global inner_p=p[-15/1000,35/1000,0,0,0,0]
          else:
            $ 2134 "Else" "noBreak"
            $ 2135 "inner_p≔p[0,0,0,0,0,0]"
            global inner_p=p[0,0,0,0,0,0]
          end
          $ 2136 "j_tp≔get_inverse_kin(pose_add(b_touch_pos,inner_p),qnear=right_j)"
          global j_tp= get_inverse_kin ( pose_add (b_touch_pos,inner_p),qnear=right_j)
        end
        $ 2137 "j_cp[0]=j_tp[0]"
        j_cp[0]=j_tp[0]
        $ 2138 "j_cp[1]=j_cp[1]+(j_tp[1]-j_cp[1])/2"
        j_cp[1]=j_cp[1]+(j_tp[1]-j_cp[1])/2
        $ 2139 "j_cp[2]=j_cp[2]+(j_tp[2]-j_cp[2])/2.5"
        j_cp[2]=j_cp[2]+(j_tp[2]-j_cp[2])/2.5
        $ 2140 "j_cp[3]=j_cp[3]+(j_tp[3]-j_cp[3])/2.5"
        j_cp[3]=j_cp[3]+(j_tp[3]-j_cp[3])/2.5
        $ 2141 "j_cp[4]=j_cp[4]+(j_tp[4]-j_cp[4])/3"
        j_cp[4]=j_cp[4]+(j_tp[4]-j_cp[4])/3
        $ 2142 "j_cp[5]=j_cp[5]+(j_tp[5]-j_cp[5])/1"
        j_cp[5]=j_cp[5]+(j_tp[5]-j_cp[5])/1
        $ 2143 "MoveJ"
        $ 2144 "j_cp" "breakAfter"
        movej(j_cp, a=1.3962634015954636, v=1.0471975511965976)
        $ 2145 "j_tp≔[j_cp[0],j_cp[1],j_cp[2],j_cp[3],j_tp[4],j_tp[5]]"
        global j_tp=[j_cp[0],j_cp[1],j_cp[2],j_cp[3],j_tp[4],j_tp[5]]
      end
      $ 2148 "If (b2_left_par≟ True ) and (b1_cell_info_L≟A or b1_cell_info_L≟C or b1_cell_info_L≟c) and (A_sel_v≠A_VL2)"
      if ((b2_left_par ==   True  )  and  (b1_cell_info_L == A  or  b1_cell_info_L == C  or  b1_cell_info_L == c)  and  (A_sel_v != A_VL2)):
        $ 2149 "begin_3f_p≔pose_trans(A_Touch_p[A_sel_v],p[(multi_offset_z*(multi_path-1))/1000,0,0,0,0,0])"
        global begin_3f_p= pose_trans (A_Touch_p[A_sel_v],p[(multi_offset_z*(multi_path-1))/1000,0,0,0,0,0])
      else:
        $ 2150 "ElseIf (b2_left_par≟ False ) and (b1_cell_info_R≟A or b1_cell_info_R≟C or b1_cell_info_R≟c) and (A_sel_v≠A_VR2)"
        if ((b2_left_par ==   False  )  and  (b1_cell_info_R == A  or  b1_cell_info_R == C  or  b1_cell_info_R == c)  and  (A_sel_v != A_VR2)):
          $ 2151 "begin_3f_p≔pose_trans(A_Touch_p[A_sel_v],p[(multi_offset_z*(multi_path-1))/1000,0,0,0,0,0])"
          global begin_3f_p= pose_trans (A_Touch_p[A_sel_v],p[(multi_offset_z*(multi_path-1))/1000,0,0,0,0,0])
        else:
          $ 2152 "Else" "noBreak"
          $ 2153 "begin_3f_p≔A_Touch_p[A_sel_v]"
          global begin_3f_p=A_Touch_p[A_sel_v]
        end
      end
      $ 2154 "If b2_left_par≟ False "
      if (b2_left_par ==   False  ):
        $ 2155 "If (b1_cell_info_R≟c or b1_cell_info_R≟d) and A_sel_v≟A_VR2"
        if ((b1_cell_info_R == c  or  b1_cell_info_R == d)  and  A_sel_v == A_VR2):
          $ 2157 "b7_tilt_degree≔[-72,-20,15]"
          global b7_tilt_degree=[-72,-20,15]
          $ 2158 "begin_3f_p=pose_add(begin_3f_p,p[-6/1000,-1.5/1000,0,0,0,0])"
          begin_3f_p= pose_add (begin_3f_p,p[-6/1000,-1.5/1000,0,0,0,0])
          $ 2159 "a2_speed_cpm≔a2_speed_cpm*1"
          global a2_speed_cpm=a2_speed_cpm*1
          $ 2160 "a3_wv_amplitude≔a3_wv_amplitude*1"
          global a3_wv_amplitude=a3_wv_amplitude*1
          $ 2161 "a4_wv_frequency≔a4_wv_frequency*1"
          global a4_wv_frequency=a4_wv_frequency*1
          $ 2162 "b3_dealy_all≔[0,b4_wv_delay2*1,0,b6_wv_delay4*1]"
          global b3_dealy_all=[0,b4_wv_delay2*1,0,b6_wv_delay4*1]
          $ 2163 "a0_volt_ref≔a0_volt_ref*1"
          global a0_volt_ref=a0_volt_ref*1
          $ 2164 "a1_amp_ref≔a1_amp_ref*1"
          global a1_amp_ref=a1_amp_ref*1
          $ 2165 "volt and current"
          $ 2166 "squash_l≔[a0_volt_ref,a1_amp_ref,squash_enable,squash_voltage,squash_current,squash_amp,squash_speed,squash_cycle,waste_cycle,c0_offset_x,c0_offset_z]"
          global squash_l=[a0_volt_ref,a1_amp_ref,squash_enable,squash_voltage,squash_current,squash_amp,squash_speed,squash_cycle,waste_cycle,c0_offset_x,c0_offset_z]
          $ 2167 "set_current_voltage(a1_amp_ref,a0_volt_ref)"
          set_current_voltage(a1_amp_ref,a0_volt_ref)
        end
      end
      $ 2176 "welding_result = line_weaving_tp(begin_3f_p,A_Touch_p[A_sel_v_end],[a8_wv_distance,Circle_Speed,b1_appro_param,a4_wv_frequency,a3_wv_amplitude,b8_wv_type,wv_direction,current_path,c8_arc_cur_offs],b7_tilt_degree,b3_dealy_all,a9_wv_weldingon,c3_wv_arc,c7_wv_gap,a5_f_hole,b8_wv_2f,a7_weld_crater,squash_l)"
      welding_result = line_weaving_tp(begin_3f_p,A_Touch_p[A_sel_v_end],[a8_wv_distance,Circle_Speed,b1_appro_param,a4_wv_frequency,a3_wv_amplitude,b8_wv_type,wv_direction,current_path,c8_arc_cur_offs],b7_tilt_degree,b3_dealy_all,a9_wv_weldingon,c3_wv_arc,c7_wv_gap,a5_f_hole,b8_wv_2f,a7_weld_crater,squash_l)
      thread_flag_2118 = 1
    end
    if (running_trig ==   True  ):
      global thread_handler_2118=run Thread_if_2118()
      while (thread_flag_2118 == 0):
        if not(running_trig ==   True  ):
          kill thread_handler_2118
          thread_flag_2118 = 2
        else:
          sync()
        end
      end
    else:
      thread_flag_2118 = 2
    end
    $ 2177 "write_port_register(weld_done_137,1)"
    write_port_register(weld_done_137,1)
    $ 2178 "homeing()"
    homeing()
    $ 2179 "If sludge≟1"
    if (sludge == 1):
      $ 2180 "pause_trig≔ True "
      global pause_trig=  True
    end
  end
  def weav_welding_2f():
    $ 2181 "weav_welding_2f" "noBreak"
    $ 2182 "If running_trig≟ True "
    global thread_flag_2182=0
    thread Thread_if_2182():
      $ 2183 "Calculation"
      $ 2184 "If Auto_W_num[Auto_cur_cell]≟31 or Auto_W_num[Auto_cur_cell]≟32 or Auto_W_num[Auto_cur_cell]≟30"
      if (Auto_W_num[Auto_cur_cell] == 31  or  Auto_W_num[Auto_cur_cell] == 32  or  Auto_W_num[Auto_cur_cell] == 30):
        $ 2185 "cal_single"
        $ 2186 "pos_m_path≔A_Touch_p[A_HOR]"
        global pos_m_path=A_Touch_p[A_HOR]
        $ 2187 "pos_m_path_end≔A_Touch_p[A_HOR_R]"
        global pos_m_path_end=A_Touch_p[A_HOR_R]
        $ 2188 "A_middle_weld≔interpolate_pose(pos_m_path, pos_m_path_end,0.5)"
        global A_middle_weld= interpolate_pose (pos_m_path, pos_m_path_end,0.5)
        $ 2189 "A_middle_weld[2]=A_touch_bottom[2]"
        A_middle_weld[2]=A_touch_bottom[2]
        $ 2190 "A_middle_weld≔p[A_middle_weld[0],A_middle_weld[1],A_middle_weld[2],pos_m_path[3],pos_m_path[4],pos_m_path[5]]"
        global A_middle_weld=p[A_middle_weld[0],A_middle_weld[1],A_middle_weld[2],pos_m_path[3],pos_m_path[4],pos_m_path[5]]
      else:
        $ 2191 "Else" "noBreak"
        $ 2193 "side_offset≔0"
        global side_offset=0
        $ 2194 "If current_path≟2 or current_path≟4"
        if (current_path == 2  or  current_path == 4):
          $ 2196 "center_offset≔0"
          global center_offset=0
        else:
          $ 2197 "Else" "noBreak"
          $ 2198 "center_offset≔0"
          global center_offset=0
        end
        $ 2199 "cal_multi"
        $ 2200 "pos_m_path≔A_Touch_p[A_HOR]"
        global pos_m_path=A_Touch_p[A_HOR]
        $ 2202 "pos_m_path_end≔A_Touch_p[A_HOR_R]"
        global pos_m_path_end=A_Touch_p[A_HOR_R]
        $ 2204 "A_middle_weld≔interpolate_pose(pos_m_path, pos_m_path_end,0.5)"
        global A_middle_weld= interpolate_pose (pos_m_path, pos_m_path_end,0.5)
        $ 2205 "A_middle_weld[2]=A_touch_bottom[2]"
        A_middle_weld[2]=A_touch_bottom[2]
        $ 2207 "A_middle_weld≔p[A_middle_weld[0],A_middle_weld[1],A_middle_weld[2],pos_m_path[3],pos_m_path[4],pos_m_path[5]]"
        global A_middle_weld=p[A_middle_weld[0],A_middle_weld[1],A_middle_weld[2],pos_m_path[3],pos_m_path[4],pos_m_path[5]]
      end
      $ 2208 "gap_half"
      $ 2209 "gap_amp_bak≔c5_wv_gap_y"
      global gap_amp_bak=c5_wv_gap_y
      $ 2210 "gap_speed_bak≔c6_wv_gap_cpm"
      global gap_speed_bak=c6_wv_gap_cpm
      $ 2211 "gap_freq_bak≔c9_wv_gap_freq"
      global gap_freq_bak=c9_wv_gap_freq
      $ 2212 "c5_wv_gap_y≔(a3_wv_amplitude+c5_wv_gap_y)/2"
      global c5_wv_gap_y=(a3_wv_amplitude+c5_wv_gap_y)/2
      $ 2213 "c6_wv_gap_cpm≔(a2_speed_cpm+c6_wv_gap_cpm)/2"
      global c6_wv_gap_cpm=(a2_speed_cpm+c6_wv_gap_cpm)/2
      $ 2214 "c9_wv_gap_freq≔(a4_wv_frequency+c9_wv_gap_freq)/2"
      global c9_wv_gap_freq=(a4_wv_frequency+c9_wv_gap_freq)/2
      $ 2215 "c7_wv_gap≔[c4_gap_enable,c5_wv_gap_y,c6_wv_gap_cpm,c9_wv_gap_freq]"
      global c7_wv_gap=[c4_gap_enable,c5_wv_gap_y,c6_wv_gap_cpm,c9_wv_gap_freq]
      $ 2216 "Weaving"
      $ 2217 "If EXT_flag1[6]"
      if (EXT_flag1[6]):
        $ 2218 "If Auto_W_num[Auto_cur_cell]%10≟1"
        if (Auto_W_num[Auto_cur_cell]%10 == 1):
          $ 2219 "inv_inching(inv_inch_time)"
          inv_inching(inv_inch_time)
          $ 2220 "wv_direction≔1"
          global wv_direction=1
          $ 2222 "step_2f≔1"
          global step_2f=1
          $ 2223 "welding_result = line_weaving_tp(A_middle_weld,pos_m_path,[a8_wv_distance,Circle_Speed,b1_appro_param,a4_wv_frequency,a3_wv_amplitude,b8_wv_type,wv_direction,current_path,c8_arc_cur_offs],b7_tilt_degree,b3_dealy_all,a9_wv_weldingon,c3_wv_arc,c7_wv_gap,a5_f_hole,b8_wv_2f,a7_weld_crater,squash_l)"
          welding_result = line_weaving_tp(A_middle_weld,pos_m_path,[a8_wv_distance,Circle_Speed,b1_appro_param,a4_wv_frequency,a3_wv_amplitude,b8_wv_type,wv_direction,current_path,c8_arc_cur_offs],b7_tilt_degree,b3_dealy_all,a9_wv_weldingon,c3_wv_arc,c7_wv_gap,a5_f_hole,b8_wv_2f,a7_weld_crater,squash_l)
          $ 2225 "Wait: 0.5"
          sleep(0.5)
        end
        $ 2226 "If Auto_W_num[Auto_cur_cell]%10≟2"
        if (Auto_W_num[Auto_cur_cell]%10 == 2):
          $ 2227 "inv_inching(inv_inch_time)"
          inv_inching(inv_inch_time)
          $ 2228 "a7_weld_crater≔[d_start_current,d_start_voltage,d_start_time,d_end_current_2,d_end_voltage_2,d_end_time_2,d_lean_degree]"
          global a7_weld_crater=[d_start_current,d_start_voltage,d_start_time,d_end_current_2,d_end_voltage_2,d_end_time_2,d_lean_degree]
          $ 2229 "gap_half_right"
          $ 2230 "a3_wv_amplitude≔gap_amp_bak"
          global a3_wv_amplitude=gap_amp_bak
          $ 2231 "a2_speed_cpm≔gap_speed_bak"
          global a2_speed_cpm=gap_speed_bak
          $ 2232 "a4_wv_frequency≔gap_freq_bak"
          global a4_wv_frequency=gap_freq_bak
          $ 2233 "c7_wv_gap≔[c4_gap_enable,c5_wv_gap_y,c6_wv_gap_cpm,c9_wv_gap_freq]"
          global c7_wv_gap=[c4_gap_enable,c5_wv_gap_y,c6_wv_gap_cpm,c9_wv_gap_freq]
          $ 2234 "wv_direction≔-1"
          global wv_direction=-1
          $ 2236 "step_2f≔2"
          global step_2f=2
          $ 2238 "welding_result = line_weaving_tp(A_middle_weld,pos_m_path_end,[a8_wv_distance,Circle_Speed,b1_appro_param,a4_wv_frequency,a3_wv_amplitude,b8_wv_type,wv_direction,current_path,c8_arc_cur_offs],b7_tilt_degree,b3_dealy_all,a9_wv_weldingon,c3_wv_arc,c7_wv_gap,a5_f_hole,b8_wv_2f,a7_weld_crater,squash_l)"
          welding_result = line_weaving_tp(A_middle_weld,pos_m_path_end,[a8_wv_distance,Circle_Speed,b1_appro_param,a4_wv_frequency,a3_wv_amplitude,b8_wv_type,wv_direction,current_path,c8_arc_cur_offs],b7_tilt_degree,b3_dealy_all,a9_wv_weldingon,c3_wv_arc,c7_wv_gap,a5_f_hole,b8_wv_2f,a7_weld_crater,squash_l)
        end
      else:
        $ 2240 "Else" "noBreak"
        $ 2241 "If Auto_W_num[Auto_cur_cell]%10≟0"
        if (Auto_W_num[Auto_cur_cell]%10 == 0):
          $ 2242 "inv_inching(inv_inch_time)"
          inv_inching(inv_inch_time)
          $ 2243 "wv_direction≔1"
          global wv_direction=1
          $ 2244 "step_2f≔1"
          global step_2f=1
          $ 2245 "welding_result = line_weaving_tp(pos_m_path,pos_m_path_end,[a8_wv_distance,Circle_Speed,b1_appro_param,a4_wv_frequency,a3_wv_amplitude,b8_wv_type,wv_direction,current_path,c8_arc_cur_offs],b7_tilt_degree,b3_dealy_all,a9_wv_weldingon,c3_wv_arc,c7_wv_gap,a5_f_hole,b8_wv_2f,a7_weld_crater,squash_l)"
          welding_result = line_weaving_tp(pos_m_path,pos_m_path_end,[a8_wv_distance,Circle_Speed,b1_appro_param,a4_wv_frequency,a3_wv_amplitude,b8_wv_type,wv_direction,current_path,c8_arc_cur_offs],b7_tilt_degree,b3_dealy_all,a9_wv_weldingon,c3_wv_arc,c7_wv_gap,a5_f_hole,b8_wv_2f,a7_weld_crater,squash_l)
        else:
          $ 2246 "Else" "noBreak"
          $ 2247 "write_port_register(142,142)"
          write_port_register(142,142)
          $ 2248 "Halt"
          halt
        end
      end
      thread_flag_2182 = 1
    end
    if (running_trig ==   True  ):
      global thread_handler_2182=run Thread_if_2182()
      while (thread_flag_2182 == 0):
        if not(running_trig ==   True  ):
          kill thread_handler_2182
          thread_flag_2182 = 2
        else:
          sync()
        end
      end
    else:
      thread_flag_2182 = 2
    end
    $ 2249 "write_port_register(weld_done_137,1)"
    write_port_register(weld_done_137,1)
    $ 2250 "MoveL"
    $ 2251 "Direction: Tool Z-"
    global move_thread_flag_2251=0
    thread move_thread_2251():
      enter_critical
      move_thread_flag_2251 = 1
      local towardsPos=calculate_point_to_move_towards(get_forward_kin(), [0.0,0.0,-1.0], 0.03)
      movel(towardsPos, a=1.2, v=0.25)
      move_thread_flag_2251 = 2
      exit_critical
    end
    move_thread_flag_2251 = 0
    move_thread_han_2251 = run move_thread_2251()
    while (True):
      sleep(1.0E-10)
      if (move_thread_flag_2251 > 1):
        join move_thread_han_2251
        $ 2252 "Until (distance)"
        break
      end
      sync()
    end
    $ 2253 "homeing()"
    homeing()
    $ 2254 "If sludge≟1 or (sludge≟2 and current_path>1)"
    if (sludge == 1  or  (sludge == 2  and  current_path>1)):
      $ 2255 "If  not (Auto_W_num[Auto_cur_cell]%10≟1)"
      if (  not  (Auto_W_num[Auto_cur_cell]%10 == 1)):
        $ 2256 "pause_trig≔ True "
        global pause_trig=  True
      end
    end
  end
  def weav_welding_2f_CD():
    $ 2257 "weav_welding_2f_CD" "noBreak"
    $ 2258 "If running_trig≟ True "
    global thread_flag_2258=0
    thread Thread_if_2258():
      $ 2259 "CD_calculation"
      $ 2260 "If (Auto_W_num[Auto_cur_cell]≥100 and Auto_W_num[Auto_cur_cell]<106)  or (Auto_W_num[Auto_cur_cell]≥150 and Auto_W_num[Auto_cur_cell]<156)"
      if ((Auto_W_num[Auto_cur_cell] >= 100  and  Auto_W_num[Auto_cur_cell]<106)   or  (Auto_W_num[Auto_cur_cell] >= 150  and  Auto_W_num[Auto_cur_cell]<156)):
        $ 2261 "cal single"
        $ 2262 "cal_1"
        $ 2263 "pos_m_path_cd≔A_Touch_p[A_sel_v]"
        global pos_m_path_cd=A_Touch_p[A_sel_v]
        $ 2264 "pos_m_p_end_cd≔A_Touch_p[A_sel_v_end]"
        global pos_m_p_end_cd=A_Touch_p[A_sel_v_end]
        $ 2265 "cal_2"
        $ 2266 "pos_m_path≔A_Touch_p[A_sel_v2]"
        global pos_m_path=A_Touch_p[A_sel_v2]
        $ 2267 "pos_m_path_end≔A_Touch_p[A_sel_v_end2]"
        global pos_m_path_end=A_Touch_p[A_sel_v_end2]
        $ 2268 "A_middle_weld≔interpolate_pose(pos_m_path, pos_m_path_end,0.5)"
        global A_middle_weld= interpolate_pose (pos_m_path, pos_m_path_end,0.5)
        $ 2269 "A_middle_weld[2]=A_touch_bottom[2]"
        A_middle_weld[2]=A_touch_bottom[2]
        $ 2270 "A_middle_weld≔p[A_middle_weld[0],A_middle_weld[1],A_middle_weld[2],pos_m_path[3],pos_m_path[4],pos_m_path[5]]"
        global A_middle_weld=p[A_middle_weld[0],A_middle_weld[1],A_middle_weld[2],pos_m_path[3],pos_m_path[4],pos_m_path[5]]
      else:
        $ 2271 "Else" "noBreak"
        $ 2272 "cal multi"
        $ 2273 "side_offset≔0"
        global side_offset=0
        $ 2274 "If current_path≟2 or current_path≟4"
        if (current_path == 2  or  current_path == 4):
          $ 2276 "center_offset≔0"
          global center_offset=0
        else:
          $ 2277 "Else" "noBreak"
          $ 2278 "center_offset≔0"
          global center_offset=0
        end
        $ 2279 "cal_1_multi"
        $ 2280 "pos_m_path_cd≔A_Touch_p[A_sel_v]"
        global pos_m_path_cd=A_Touch_p[A_sel_v]
        $ 2282 "pos_m_p_end_cd≔A_Touch_p[A_sel_v_end]"
        global pos_m_p_end_cd=A_Touch_p[A_sel_v_end]
        $ 2284 "cal_2_multi"
        $ 2285 "pos_m_path≔A_Touch_p[A_sel_v2]"
        global pos_m_path=A_Touch_p[A_sel_v2]
        $ 2287 "pos_m_path_end≔A_Touch_p[A_sel_v_end2]"
        global pos_m_path_end=A_Touch_p[A_sel_v_end2]
        $ 2289 "A_middle_weld≔interpolate_pose(pos_m_path, pos_m_path_end,0.5)"
        global A_middle_weld= interpolate_pose (pos_m_path, pos_m_path_end,0.5)
        $ 2290 "A_middle_weld[2]=A_touch_bottom[2]"
        A_middle_weld[2]=A_touch_bottom[2]
        $ 2292 "A_middle_weld≔p[A_middle_weld[0],A_middle_weld[1],A_middle_weld[2],pos_m_path[3],pos_m_path[4],pos_m_path[5]]"
        global A_middle_weld=p[A_middle_weld[0],A_middle_weld[1],A_middle_weld[2],pos_m_path[3],pos_m_path[4],pos_m_path[5]]
      end
      $ 2293 "gap_half"
      $ 2294 "gap_amp_bak≔c5_wv_gap_y"
      global gap_amp_bak=c5_wv_gap_y
      $ 2295 "gap_speed_bak≔c6_wv_gap_cpm"
      global gap_speed_bak=c6_wv_gap_cpm
      $ 2296 "gap_freq_bak≔c9_wv_gap_freq"
      global gap_freq_bak=c9_wv_gap_freq
      $ 2297 "c5_wv_gap_y≔(a3_wv_amplitude+c5_wv_gap_y)/2"
      global c5_wv_gap_y=(a3_wv_amplitude+c5_wv_gap_y)/2
      $ 2298 "c6_wv_gap_cpm≔(a2_speed_cpm+c6_wv_gap_cpm)/2"
      global c6_wv_gap_cpm=(a2_speed_cpm+c6_wv_gap_cpm)/2
      $ 2299 "c9_wv_gap_freq≔(a4_wv_frequency+c9_wv_gap_freq)/2"
      global c9_wv_gap_freq=(a4_wv_frequency+c9_wv_gap_freq)/2
      $ 2300 "c7_wv_gap≔[c4_gap_enable,c5_wv_gap_y,c6_wv_gap_cpm,c9_wv_gap_freq]"
      global c7_wv_gap=[c4_gap_enable,c5_wv_gap_y,c6_wv_gap_cpm,c9_wv_gap_freq]
      $ 2301 "If EXT_flag1[4]≟ True  and (b1_cell_info_L≠c and b1_cell_info_L≠d and b1_cell_info_R≠c and b1_cell_info_R≠d)"
      if (EXT_flag1[4] ==   True    and  (b1_cell_info_L != c  and  b1_cell_info_L != d  and  b1_cell_info_R != c  and  b1_cell_info_R != d)):
        $ 2302 "If EXT_flag1[6]"
        if (EXT_flag1[6]):
          $ 2303 "If Auto_W_num[Auto_cur_cell]%10≟1"
          if (Auto_W_num[Auto_cur_cell]%10 == 1):
            $ 2304 "inv_inching(inv_inch_time)"
            inv_inching(inv_inch_time)
            $ 2305 "step_2f≔1"
            global step_2f=1
            $ 2306 "welding_result = line_weaving_tp_l(pos_m_path_cd,[pos_m_p_end_cd,pos_m_path,A_middle_weld],[a8_wv_distance,Circle_Speed,b1_appro_param,a4_wv_frequency,a3_wv_amplitude,b8_wv_type,wv_direction,current_path,c8_arc_cur_offs],b7_tilt_degree,b3_dealy_all,a9_wv_weldingon,c3_wv_arc,c7_wv_gap,a5_f_hole,b8_wv_2f,a7_weld_crater,squash_l)"
            welding_result = line_weaving_tp_l(pos_m_path_cd,[pos_m_p_end_cd,pos_m_path,A_middle_weld],[a8_wv_distance,Circle_Speed,b1_appro_param,a4_wv_frequency,a3_wv_amplitude,b8_wv_type,wv_direction,current_path,c8_arc_cur_offs],b7_tilt_degree,b3_dealy_all,a9_wv_weldingon,c3_wv_arc,c7_wv_gap,a5_f_hole,b8_wv_2f,a7_weld_crater,squash_l)
          end
          $ 2307 "If Auto_W_num[Auto_cur_cell]%10≟4"
          if (Auto_W_num[Auto_cur_cell]%10 == 4):
            $ 2308 "inv_inching(inv_inch_time)"
            inv_inching(inv_inch_time)
            $ 2309 "a7_weld_crater≔[d_start_current,d_start_voltage,d_start_time,d_end_current_2,d_end_voltage_2,d_end_time_2,d_lean_degree]"
            global a7_weld_crater=[d_start_current,d_start_voltage,d_start_time,d_end_current_2,d_end_voltage_2,d_end_time_2,d_lean_degree]
            $ 2310 "gap_half"
            $ 2311 "a3_wv_amplitude≔gap_amp_bak"
            global a3_wv_amplitude=gap_amp_bak
            $ 2312 "a2_speed_cpm≔gap_speed_bak"
            global a2_speed_cpm=gap_speed_bak
            $ 2313 "a4_wv_frequency≔gap_freq_bak"
            global a4_wv_frequency=gap_freq_bak
            $ 2314 "c7_wv_gap≔[c4_gap_enable,c5_wv_gap_y,c6_wv_gap_cpm,c9_wv_gap_freq]"
            global c7_wv_gap=[c4_gap_enable,c5_wv_gap_y,c6_wv_gap_cpm,c9_wv_gap_freq]
            $ 2315 "step_2f≔2"
            global step_2f=2
            $ 2316 "wv_direction≔-1*wv_direction"
            global wv_direction=-1*wv_direction
            $ 2318 "welding_result = line_weaving_tp(pos_m_path_end,A_middle_weld,[a8_wv_distance,Circle_Speed,b1_appro_param,a4_wv_frequency,a3_wv_amplitude,b8_wv_type,wv_direction,current_path,c8_arc_cur_offs],b7_tilt_degree,b3_dealy_all,a9_wv_weldingon,c3_wv_arc,c7_wv_gap,a5_f_hole,b8_wv_2f,a7_weld_crater,squash_l)"
            welding_result = line_weaving_tp(pos_m_path_end,A_middle_weld,[a8_wv_distance,Circle_Speed,b1_appro_param,a4_wv_frequency,a3_wv_amplitude,b8_wv_type,wv_direction,current_path,c8_arc_cur_offs],b7_tilt_degree,b3_dealy_all,a9_wv_weldingon,c3_wv_arc,c7_wv_gap,a5_f_hole,b8_wv_2f,a7_weld_crater,squash_l)
          end
        else:
          $ 2319 "Else" "noBreak"
          $ 2320 "If Auto_W_num[Auto_cur_cell]%10≟0"
          if (Auto_W_num[Auto_cur_cell]%10 == 0):
            $ 2321 "inv_inching(inv_inch_time)"
            inv_inching(inv_inch_time)
            $ 2322 "step_2f≔1"
            global step_2f=1
            $ 2323 "welding_result = line_weaving_tp_l(pos_m_path_cd,[pos_m_p_end_cd,pos_m_path,pos_m_path_end],[a8_wv_distance,Circle_Speed,b1_appro_param,a4_wv_frequency,a3_wv_amplitude,b8_wv_type,wv_direction,current_path,c8_arc_cur_offs],b7_tilt_degree,b3_dealy_all,a9_wv_weldingon,c3_wv_arc,c7_wv_gap,a5_f_hole,b8_wv_2f,a7_weld_crater,squash_l)"
            welding_result = line_weaving_tp_l(pos_m_path_cd,[pos_m_p_end_cd,pos_m_path,pos_m_path_end],[a8_wv_distance,Circle_Speed,b1_appro_param,a4_wv_frequency,a3_wv_amplitude,b8_wv_type,wv_direction,current_path,c8_arc_cur_offs],b7_tilt_degree,b3_dealy_all,a9_wv_weldingon,c3_wv_arc,c7_wv_gap,a5_f_hole,b8_wv_2f,a7_weld_crater,squash_l)
          else:
            $ 2324 "Else" "noBreak"
            $ 2325 "write_port_register(142,142)"
            write_port_register(142,142)
            $ 2326 "Halt"
            halt
          end
        end
      else:
        $ 2327 "Else" "noBreak"
        $ 2328 "If EXT_flag1[6]"
        if (EXT_flag1[6]):
          $ 2329 "If Auto_W_num[Auto_cur_cell]%10≟2"
          if (Auto_W_num[Auto_cur_cell]%10 == 2):
            $ 2330 "inv_inching(inv_inch_time)"
            inv_inching(inv_inch_time)
            $ 2331 "step_2f≔1"
            global step_2f=1
            $ 2332 "gap_half"
            $ 2333 "gap_amp_bak≔c5_wv_gap_y"
            global gap_amp_bak=c5_wv_gap_y
            $ 2334 "gap_speed_bak≔c6_wv_gap_cpm"
            global gap_speed_bak=c6_wv_gap_cpm
            $ 2335 "gap_freq_bak≔c9_wv_gap_freq"
            global gap_freq_bak=c9_wv_gap_freq
            $ 2336 "c5_wv_gap_y≔(a3_wv_amplitude+c5_wv_gap_y)/2"
            global c5_wv_gap_y=(a3_wv_amplitude+c5_wv_gap_y)/2
            $ 2337 "c6_wv_gap_cpm≔(a2_speed_cpm+c6_wv_gap_cpm)/2"
            global c6_wv_gap_cpm=(a2_speed_cpm+c6_wv_gap_cpm)/2
            $ 2338 "c9_wv_gap_freq≔(a4_wv_frequency+c9_wv_gap_freq)/2"
            global c9_wv_gap_freq=(a4_wv_frequency+c9_wv_gap_freq)/2
            $ 2339 "c7_wv_gap≔[c4_gap_enable,c5_wv_gap_y,c6_wv_gap_cpm,c9_wv_gap_freq]"
            global c7_wv_gap=[c4_gap_enable,c5_wv_gap_y,c6_wv_gap_cpm,c9_wv_gap_freq]
            $ 2340 "welding_result = line_weaving_tp(pos_m_path_cd,pos_m_p_end_cd,[a8_wv_distance,Circle_Speed,b1_appro_param,a4_wv_frequency,a3_wv_amplitude,b8_wv_type,wv_direction,current_path,c8_arc_cur_offs],b7_tilt_degree,b3_dealy_all,a9_wv_weldingon,c3_wv_arc,c7_wv_gap,a5_f_hole,b8_wv_2f,a7_weld_crater,squash_l)"
            welding_result = line_weaving_tp(pos_m_path_cd,pos_m_p_end_cd,[a8_wv_distance,Circle_Speed,b1_appro_param,a4_wv_frequency,a3_wv_amplitude,b8_wv_type,wv_direction,current_path,c8_arc_cur_offs],b7_tilt_degree,b3_dealy_all,a9_wv_weldingon,c3_wv_arc,c7_wv_gap,a5_f_hole,b8_wv_2f,a7_weld_crater,squash_l)
            $ 2341 "Wait: 0.5"
            sleep(0.5)
          end
          $ 2342 "If Auto_W_num[Auto_cur_cell]%10≟3"
          if (Auto_W_num[Auto_cur_cell]%10 == 3):
            $ 2343 "inv_inching(inv_inch_time)"
            inv_inching(inv_inch_time)
            $ 2344 "step_2f≔2"
            global step_2f=2
            $ 2345 "welding_result = line_weaving_tp(pos_m_path,A_middle_weld,[a8_wv_distance,Circle_Speed,b1_appro_param,a4_wv_frequency,a3_wv_amplitude,b8_wv_type,wv_direction,current_path,c8_arc_cur_offs],b7_tilt_degree,b3_dealy_all,a9_wv_weldingon,c3_wv_arc,c7_wv_gap,a5_f_hole,b8_wv_2f,a7_weld_crater,squash_l)"
            welding_result = line_weaving_tp(pos_m_path,A_middle_weld,[a8_wv_distance,Circle_Speed,b1_appro_param,a4_wv_frequency,a3_wv_amplitude,b8_wv_type,wv_direction,current_path,c8_arc_cur_offs],b7_tilt_degree,b3_dealy_all,a9_wv_weldingon,c3_wv_arc,c7_wv_gap,a5_f_hole,b8_wv_2f,a7_weld_crater,squash_l)
            $ 2346 "Wait: 0.5"
            sleep(0.5)
          end
          $ 2347 "If Auto_W_num[Auto_cur_cell]%10≟4"
          if (Auto_W_num[Auto_cur_cell]%10 == 4):
            $ 2348 "inv_inching(inv_inch_time)"
            inv_inching(inv_inch_time)
            $ 2349 "a7_weld_crater≔[d_start_current,d_start_voltage,d_start_time,d_end_current_2,d_end_voltage_2,d_end_time_2,d_lean_degree]"
            global a7_weld_crater=[d_start_current,d_start_voltage,d_start_time,d_end_current_2,d_end_voltage_2,d_end_time_2,d_lean_degree]
            $ 2350 "step_2f≔3"
            global step_2f=3
            $ 2351 "gap_half"
            $ 2352 "a3_wv_amplitude≔gap_amp_bak"
            global a3_wv_amplitude=gap_amp_bak
            $ 2353 "a2_speed_cpm≔gap_speed_bak"
            global a2_speed_cpm=gap_speed_bak
            $ 2354 "a4_wv_frequency≔gap_freq_bak"
            global a4_wv_frequency=gap_freq_bak
            $ 2355 "c7_wv_gap≔[c4_gap_enable,c5_wv_gap_y,c6_wv_gap_cpm,c9_wv_gap_freq]"
            global c7_wv_gap=[c4_gap_enable,c5_wv_gap_y,c6_wv_gap_cpm,c9_wv_gap_freq]
            $ 2356 "wv_direction≔-1*wv_direction"
            global wv_direction=-1*wv_direction
            $ 2358 "welding_result = line_weaving_tp(pos_m_path_end,A_middle_weld,[a8_wv_distance,Circle_Speed,b1_appro_param,a4_wv_frequency,a3_wv_amplitude,b8_wv_type,wv_direction,current_path,c8_arc_cur_offs],b7_tilt_degree,b3_dealy_all,a9_wv_weldingon,c3_wv_arc,c7_wv_gap,a5_f_hole,b8_wv_2f,a7_weld_crater,squash_l)"
            welding_result = line_weaving_tp(pos_m_path_end,A_middle_weld,[a8_wv_distance,Circle_Speed,b1_appro_param,a4_wv_frequency,a3_wv_amplitude,b8_wv_type,wv_direction,current_path,c8_arc_cur_offs],b7_tilt_degree,b3_dealy_all,a9_wv_weldingon,c3_wv_arc,c7_wv_gap,a5_f_hole,b8_wv_2f,a7_weld_crater,squash_l)
          end
        else:
          $ 2359 "Else" "noBreak"
          $ 2360 "If Auto_W_num[Auto_cur_cell]%10≟2"
          if (Auto_W_num[Auto_cur_cell]%10 == 2):
            $ 2361 "inv_inching(inv_inch_time)"
            inv_inching(inv_inch_time)
            $ 2362 "step_2f≔1"
            global step_2f=1
            $ 2363 "c7_wv_gap≔[0,c5_wv_gap_y,c6_wv_gap_cpm,c9_wv_gap_freq]"
            global c7_wv_gap=[0,c5_wv_gap_y,c6_wv_gap_cpm,c9_wv_gap_freq]
            $ 2364 "welding_result = line_weaving_tp(pos_m_path_cd,pos_m_p_end_cd,[a8_wv_distance,Circle_Speed,b1_appro_param,a4_wv_frequency,a3_wv_amplitude,b8_wv_type,wv_direction,current_path,c8_arc_cur_offs],b7_tilt_degree,b3_dealy_all,a9_wv_weldingon,c3_wv_arc,c7_wv_gap,a5_f_hole,b8_wv_2f,a7_weld_crater,squash_l)"
            welding_result = line_weaving_tp(pos_m_path_cd,pos_m_p_end_cd,[a8_wv_distance,Circle_Speed,b1_appro_param,a4_wv_frequency,a3_wv_amplitude,b8_wv_type,wv_direction,current_path,c8_arc_cur_offs],b7_tilt_degree,b3_dealy_all,a9_wv_weldingon,c3_wv_arc,c7_wv_gap,a5_f_hole,b8_wv_2f,a7_weld_crater,squash_l)
            $ 2365 "Wait: 0.5"
            sleep(0.5)
          end
          $ 2366 "If Auto_W_num[Auto_cur_cell]%10≟5"
          if (Auto_W_num[Auto_cur_cell]%10 == 5):
            $ 2367 "inv_inching(inv_inch_time)"
            inv_inching(inv_inch_time)
            $ 2368 "step_2f≔2"
            global step_2f=2
            $ 2369 "c7_wv_gap≔[c4_gap_enable,c5_wv_gap_y,c6_wv_gap_cpm,c9_wv_gap_freq]"
            global c7_wv_gap=[c4_gap_enable,c5_wv_gap_y,c6_wv_gap_cpm,c9_wv_gap_freq]
            $ 2370 "welding_result = line_weaving_tp(pos_m_path,pos_m_path_end,[a8_wv_distance,Circle_Speed,b1_appro_param,a4_wv_frequency,a3_wv_amplitude,b8_wv_type,wv_direction,current_path,c8_arc_cur_offs],b7_tilt_degree,b3_dealy_all,a9_wv_weldingon,c3_wv_arc,c7_wv_gap,a5_f_hole,b8_wv_2f,a7_weld_crater,squash_l)"
            welding_result = line_weaving_tp(pos_m_path,pos_m_path_end,[a8_wv_distance,Circle_Speed,b1_appro_param,a4_wv_frequency,a3_wv_amplitude,b8_wv_type,wv_direction,current_path,c8_arc_cur_offs],b7_tilt_degree,b3_dealy_all,a9_wv_weldingon,c3_wv_arc,c7_wv_gap,a5_f_hole,b8_wv_2f,a7_weld_crater,squash_l)
            $ 2371 "Wait: 0.5"
            sleep(0.5)
          end
        end
      end
      thread_flag_2258 = 1
    end
    if (running_trig ==   True  ):
      global thread_handler_2258=run Thread_if_2258()
      while (thread_flag_2258 == 0):
        if not(running_trig ==   True  ):
          kill thread_handler_2258
          thread_flag_2258 = 2
        else:
          sync()
        end
      end
    else:
      thread_flag_2258 = 2
    end
    $ 2372 "write_port_register(weld_done_137,1)"
    write_port_register(weld_done_137,1)
    $ 2376 "wv_direction≔1"
    global wv_direction=1
    $ 2377 "If Auto_W_num[Auto_cur_cell]≥150"
    if (Auto_W_num[Auto_cur_cell] >= 150):
      $ 2378 "MoveL"
      $ 2379 "Direction: Base"
      global move_thread_flag_2379=0
      thread move_thread_2379():
        enter_critical
        move_thread_flag_2379 = 1
        local towardsPos=calculate_point_to_move_towards(p[0.0,0.0,0.0,0.0,0.0,0.0], [-1,1,0.0], 0.03)
        movel(towardsPos, a=0.2, v=0.05)
        move_thread_flag_2379 = 2
        exit_critical
      end
      move_thread_flag_2379 = 0
      move_thread_han_2379 = run move_thread_2379()
      while (True):
        sleep(1.0E-10)
        if (move_thread_flag_2379 > 1):
          join move_thread_han_2379
          $ 2380 "Until (distance)"
          break
        end
        sync()
      end
    else:
      $ 2381 "ElseIf Auto_W_num[Auto_cur_cell]≥100"
      if (Auto_W_num[Auto_cur_cell] >= 100):
        $ 2382 "MoveL"
        $ 2383 "Direction: Base"
        global move_thread_flag_2383=0
        thread move_thread_2383():
          enter_critical
          move_thread_flag_2383 = 1
          local towardsPos=calculate_point_to_move_towards(p[0.0,0.0,0.0,0.0,0.0,0.0], [-1,-1,0.0], 0.03)
          movel(towardsPos, a=0.2, v=0.05)
          move_thread_flag_2383 = 2
          exit_critical
        end
        move_thread_flag_2383 = 0
        move_thread_han_2383 = run move_thread_2383()
        while (True):
          sleep(1.0E-10)
          if (move_thread_flag_2383 > 1):
            join move_thread_han_2383
            $ 2384 "Until (distance)"
            break
          end
          sync()
        end
      end
    end
    $ 2385 "MoveL"
    $ 2386 "Direction: Tool Z-"
    global move_thread_flag_2386=0
    thread move_thread_2386():
      enter_critical
      move_thread_flag_2386 = 1
      local towardsPos=calculate_point_to_move_towards(get_forward_kin(), [0.0,0.0,-1.0], 0.03)
      movel(towardsPos, a=1.2, v=0.25)
      move_thread_flag_2386 = 2
      exit_critical
    end
    move_thread_flag_2386 = 0
    move_thread_han_2386 = run move_thread_2386()
    while (True):
      sleep(1.0E-10)
      if (move_thread_flag_2386 > 1):
        join move_thread_han_2386
        $ 2387 "Until (distance)"
        break
      end
      sync()
    end
    $ 2388 "homeing()"
    homeing()
    $ 2389 "If sludge≟1 or (sludge≟2 and current_path>1)"
    if (sludge == 1  or  (sludge == 2  and  current_path>1)):
      $ 2390 "If  not (Auto_W_num[Auto_cur_cell]%10≟1 or Auto_W_num[Auto_cur_cell]%10≟2 or Auto_W_num[Auto_cur_cell]%10≟3)"
      if (  not  (Auto_W_num[Auto_cur_cell]%10 == 1  or  Auto_W_num[Auto_cur_cell]%10 == 2  or  Auto_W_num[Auto_cur_cell]%10 == 3)):
        $ 2391 "pause_trig≔ True "
        global pause_trig=  True
      end
    end
  end
  def reset_weld_param():
    $ 2392 "reset_weld_param" "noBreak"
    $ 2393 "start_num≔225"
    global start_num=225
    $ 2394 "Loop start_num<237"
    while (start_num<237):
      $ 2395 "write_port_register(start_num,0)"
      write_port_register(start_num,0)
      $ 2396 "start_num≔start_num+1"
      global start_num=start_num+1
    end
    $ 2397 "start_num≔240"
    global start_num=240
    $ 2398 "Loop start_num<256"
    while (start_num<256):
      $ 2399 "write_port_register(start_num,0)"
      write_port_register(start_num,0)
      $ 2400 "start_num≔start_num+1"
      global start_num=start_num+1
    end
  end
  def touch_sub():
    $ 2401 "touch_sub" "noBreak"
    $ 2402 "freedrive"
    $ 2403 "save_timer: Start"
    save_timer_is_counting = True
    $ 2404 "Loop save_tool≟ False  and save_timer≤0.5"
    while (get_tool_digital_in(0) ==   False    and  save_timer <= 0.5):
      $ 2405 "If save_tool≟ False "
      if (get_tool_digital_in(0) ==   False  ):
        $ 2406 "save_timer≔0"
        global save_timer=0
      end
      $ 2407 "If freedrive≟ True  and freedrive_trg≟ False "
      if (get_tool_digital_in(1) ==   True    and  freedrive_trg ==   False  ):
        $ 2408 "'Manual - Freedrive'"
        # 'Manual - Freedrive'
        $ 2409 "freedrive_mode()"
        freedrive_mode()
        $ 2410 "freedrive_trg≔ True "
        global freedrive_trg=  True
      else:
        $ 2411 "ElseIf freedrive≟ False  and freedrive_trg≟ True "
        if (get_tool_digital_in(1) ==   False    and  freedrive_trg ==   True  ):
          $ 2412 "end_freedrive_mode()"
          end_freedrive_mode()
          $ 2413 "freedrive_trg≔ False "
          global freedrive_trg=  False
        end
      end
      $ 2414 "If lamp_trig≟ False "
      if (lamp_trig ==   False  ):
        $ 2415 "lamp_trig≔ True "
        global lamp_trig=  True
      end
      $ 2416 "sync()"
      sync()
    end
    $ 2417 "save_timer: Stop"
    save_timer_is_counting = False
    $ 2418 "save_timer: Reset"
    save_timer = 0
    $ 2419 "write_port_register(touch_done_157,1)"
    write_port_register(touch_done_157,1)
    $ 2420 "Wait read_port_register(touch_done_157)≟0"
    while (not( read_port_register (touch_done_157) == 0)):
      sync()
    end
    $ 2421 "Wait save_tool=LO"
    while (get_tool_digital_in(0) == True):
      sync()
    end
  end
  $ 2 "BeforeStart"
  $ 3 "'RobotVersion'"
  # 'RobotVersion'
  $ 4 "write_port_register(160,104)"
  write_port_register(160,104)
  $ 5 "Teaching for Touch"
  $ 6 "g_current_p≔get_actual_tcp_pose()"
  global g_current_p= get_actual_tcp_pose ()
  $ 7 "MoveJ"
  $ 8 "g_current_p" "breakAfter"
